REGION Network 14: Interface Signals 05 -Example: Model Flex-Pro-Line - IN/OUT- / Interface Signals 09
   // Aufruf des Schnittstellen Signal Bausteins Ba-Bereich 4 / Call the interface signals bool blocks of opmode 4
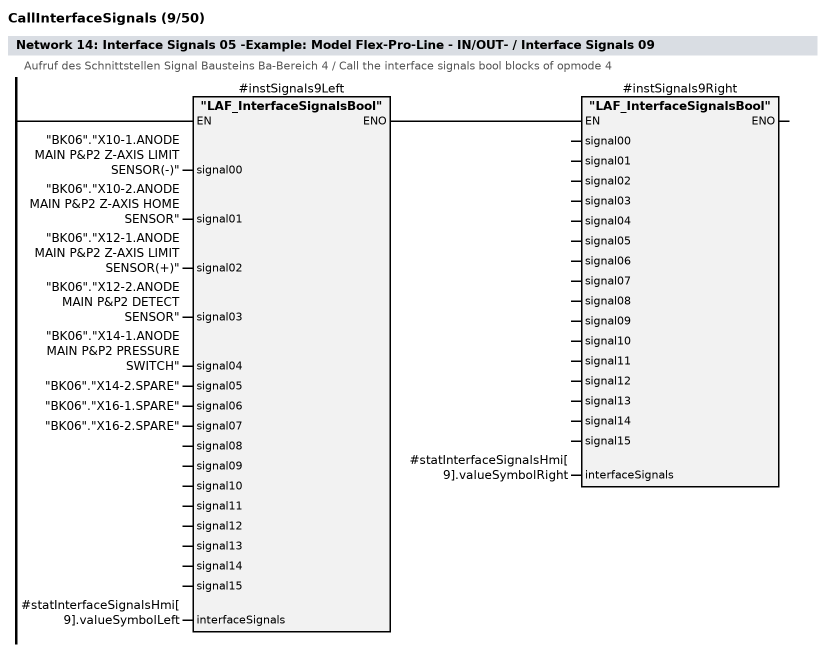
   RUNG wire#powerrail
      #instSignals9Left(signal00 := "BK06"."X10-1.ANODE MAIN P&P2 Z-AXIS LIMIT SENSOR(-)", signal01 := "BK06"."X10-2.ANODE MAIN P&P2 Z-AXIS HOME SENSOR", signal02 := "BK06"."X12-1.ANODE MAIN P&P2 Z-AXIS LIMIT SENSOR(+)", signal03 := "BK06"."X12-2.ANODE MAIN P&P2 DETECT SENSOR", signal04 := "BK06"."X14-1.ANODE MAIN P&P2 PRESSURE SWITCH", signal05 := "BK06"."X14-2.SPARE", signal06 := "BK06"."X16-1.SPARE", signal07 := "BK06"."X16-2.SPARE", signal08 :=, signal09 :=, signal10 :=, signal11 :=, signal12 :=, signal13 :=, signal14 :=, signal15 :=, interfaceSignals := #statInterfaceSignalsHmi[9].valueSymbolLeft)
      #instSignals9Right(signal00 :=, signal01 :=, signal02 :=, signal03 :=, signal04 :=, signal05 :=, signal06 :=, signal07 :=, signal08 :=, signal09 :=, signal10 :=, signal11 :=, signal12 :=, signal13 :=, signal14 :=, signal15 :=, interfaceSignals := #statInterfaceSignalsHmi[9].valueSymbolRight)
   END_RUNG
   // the same network as SCL:
   #instSignals9Left(signal00 := "BK06"."X10-1.ANODE MAIN P&P2 Z-AXIS LIMIT SENSOR(-)",   // "LAF_InterfaceSignalsBool"
                     signal01 := "BK06"."X10-2.ANODE MAIN P&P2 Z-AXIS HOME SENSOR",
                     signal02 := "BK06"."X12-1.ANODE MAIN P&P2 Z-AXIS LIMIT SENSOR(+)",
                     signal03 := "BK06"."X12-2.ANODE MAIN P&P2 DETECT SENSOR",
                     signal04 := "BK06"."X14-1.ANODE MAIN P&P2 PRESSURE SWITCH",
                     signal05 := "BK06"."X14-2.SPARE",
                     signal06 := "BK06"."X16-1.SPARE",
                     signal07 := "BK06"."X16-2.SPARE",
                     interfaceSignals := #statInterfaceSignalsHmi[9].valueSymbolLeft,
                     ENO => #_w1);
   IF #_w1 THEN
       #instSignals9Right(interfaceSignals := #statInterfaceSignalsHmi[9].valueSymbolRight);   // "LAF_InterfaceSignalsBool"
   END_IF;
END_REGION

REGION Network 15: Interface Signals 05 -Example: Model Flex-Pro-Line - IN/OUT- / Interface Signals 10
   // Aufruf des Schnittstellen Signal Bausteins Ba-Bereich 4 / Call the interface signals bool blocks of opmode 4
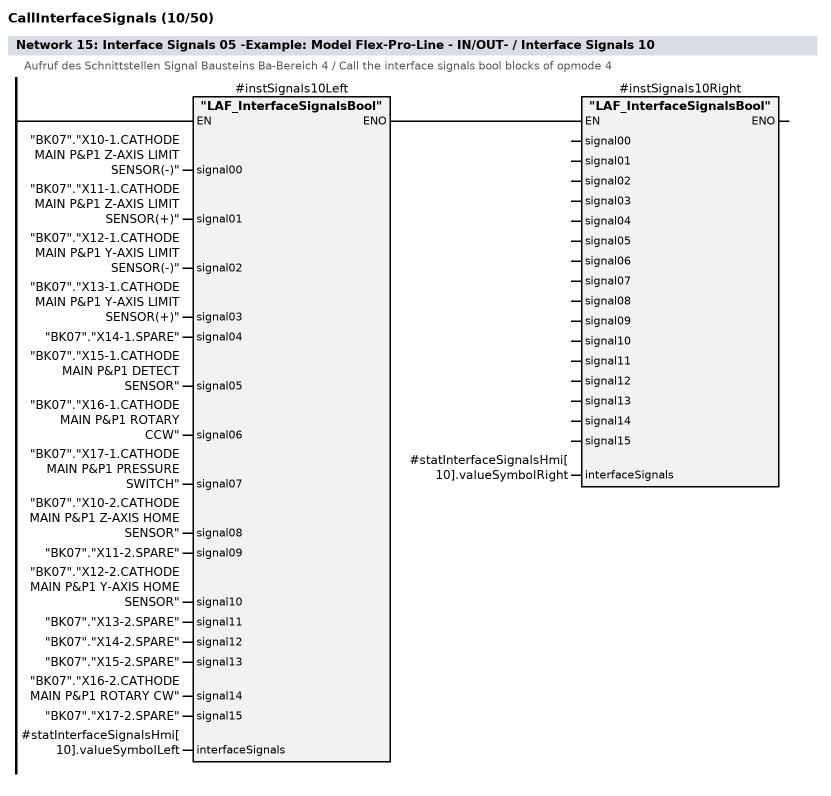
   RUNG wire#powerrail
      #instSignals10Left(signal00 := "BK07"."X10-1.CATHODE MAIN P&P1 Z-AXIS LIMIT SENSOR(-)", signal01 := "BK07"."X11-1.CATHODE MAIN P&P1 Z-AXIS LIMIT SENSOR(+)", signal02 := "BK07"."X12-1.CATHODE MAIN P&P1 Y-AXIS LIMIT SENSOR(-)", signal03 := "BK07"."X13-1.CATHODE MAIN P&P1 Y-AXIS LIMIT SENSOR(+)", signal04 := "BK07"."X14-1.SPARE", signal05 := "BK07"."X15-1.CATHODE MAIN P&P1 DETECT SENSOR", signal06 := "BK07"."X16-1.CATHODE MAIN P&P1 ROTARY CCW", signal07 := "BK07"."X17-1.CATHODE MAIN P&P1 PRESSURE SWITCH", signal08 := "BK07"."X10-2.CATHODE MAIN P&P1 Z-AXIS HOME SENSOR", signal09 := "BK07"."X11-2.SPARE", signal10 := "BK07"."X12-2.CATHODE MAIN P&P1 Y-AXIS HOME SENSOR", signal11 := "BK07"."X13-2.SPARE", signal12 := "BK07"."X14-2.SPARE", signal13 := "BK07"."X15-2.SPARE", signal14 := "BK07"."X16-2.CATHODE MAIN P&P1 ROTARY CW", signal15 := "BK07"."X17-2.SPARE", interfaceSignals := #statInterfaceSignalsHmi[10].valueSymbolLeft)
      #instSignals10Right(signal00 :=, signal01 :=, signal02 :=, signal03 :=, signal04 :=, signal05 :=, signal06 :=, signal07 :=, signal08 :=, signal09 :=, signal10 :=, signal11 :=, signal12 :=, signal13 :=, signal14 :=, signal15 :=, interfaceSignals := #statInterfaceSignalsHmi[10].valueSymbolRight)
   END_RUNG
   // the same network as SCL:
   #instSignals10Left(signal00 := "BK07"."X10-1.CATHODE MAIN P&P1 Z-AXIS LIMIT SENSOR(-)",   // "LAF_InterfaceSignalsBool"
                      signal01 := "BK07"."X11-1.CATHODE MAIN P&P1 Z-AXIS LIMIT SENSOR(+)",
                      signal02 := "BK07"."X12-1.CATHODE MAIN P&P1 Y-AXIS LIMIT SENSOR(-)",
                      signal03 := "BK07"."X13-1.CATHODE MAIN P&P1 Y-AXIS LIMIT SENSOR(+)",
                      signal04 := "BK07"."X14-1.SPARE",
                      signal05 := "BK07"."X15-1.CATHODE MAIN P&P1 DETECT SENSOR",
                      signal06 := "BK07"."X16-1.CATHODE MAIN P&P1 ROTARY CCW",
                      signal07 := "BK07"."X17-1.CATHODE MAIN P&P1 PRESSURE SWITCH",
                      signal08 := "BK07"."X10-2.CATHODE MAIN P&P1 Z-AXIS HOME SENSOR",
                      signal09 := "BK07"."X11-2.SPARE",
                      signal10 := "BK07"."X12-2.CATHODE MAIN P&P1 Y-AXIS HOME SENSOR",
                      signal11 := "BK07"."X13-2.SPARE",
                      signal12 := "BK07"."X14-2.SPARE",
                      signal13 := "BK07"."X15-2.SPARE",
                      signal14 := "BK07"."X16-2.CATHODE MAIN P&P1 ROTARY CW",
                      signal15 := "BK07"."X17-2.SPARE",
                      interfaceSignals := #statInterfaceSignalsHmi[10].valueSymbolLeft,
                      ENO => #_w1);
   IF #_w1 THEN
       #instSignals10Right(interfaceSignals := #statInterfaceSignalsHmi[10].valueSymbolRight);   // "LAF_InterfaceSignalsBool"
   END_IF;
END_REGION

REGION Network 16: Interface Signals 05 -Example: Model Flex-Pro-Line - IN/OUT- / Interface Signals 11
   // Aufruf des Schnittstellen Signal Bausteins Ba-Bereich 4 / Call the interface signals bool blocks of opmode 4
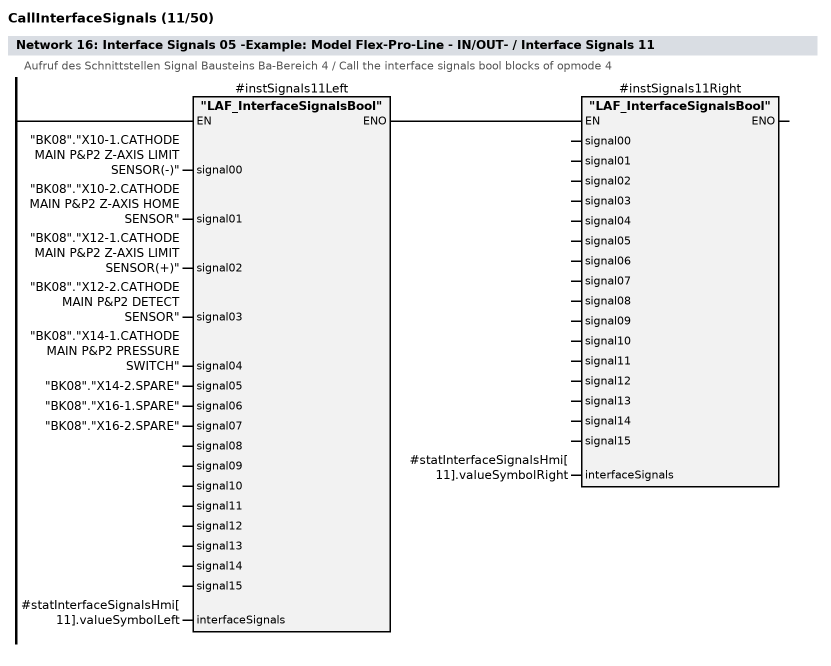
   RUNG wire#powerrail
      #instSignals11Left(signal00 := "BK08"."X10-1.CATHODE MAIN P&P2 Z-AXIS LIMIT SENSOR(-)", signal01 := "BK08"."X10-2.CATHODE MAIN P&P2 Z-AXIS HOME SENSOR", signal02 := "BK08"."X12-1.CATHODE MAIN P&P2 Z-AXIS LIMIT SENSOR(+)", signal03 := "BK08"."X12-2.CATHODE MAIN P&P2 DETECT SENSOR", signal04 := "BK08"."X14-1.CATHODE MAIN P&P2 PRESSURE SWITCH", signal05 := "BK08"."X14-2.SPARE", signal06 := "BK08"."X16-1.SPARE", signal07 := "BK08"."X16-2.SPARE", signal08 :=, signal09 :=, signal10 :=, signal11 :=, signal12 :=, signal13 :=, signal14 :=, signal15 :=, interfaceSignals := #statInterfaceSignalsHmi[11].valueSymbolLeft)
      #instSignals11Right(signal00 :=, signal01 :=, signal02 :=, signal03 :=, signal04 :=, signal05 :=, signal06 :=, signal07 :=, signal08 :=, signal09 :=, signal10 :=, signal11 :=, signal12 :=, signal13 :=, signal14 :=, signal15 :=, interfaceSignals := #statInterfaceSignalsHmi[11].valueSymbolRight)
   END_RUNG
   // the same network as SCL:
   #instSignals11Left(signal00 := "BK08"."X10-1.CATHODE MAIN P&P2 Z-AXIS LIMIT SENSOR(-)",   // "LAF_InterfaceSignalsBool"
                      signal01 := "BK08"."X10-2.CATHODE MAIN P&P2 Z-AXIS HOME SENSOR",
                      signal02 := "BK08"."X12-1.CATHODE MAIN P&P2 Z-AXIS LIMIT SENSOR(+)",
                      signal03 := "BK08"."X12-2.CATHODE MAIN P&P2 DETECT SENSOR",
                      signal04 := "BK08"."X14-1.CATHODE MAIN P&P2 PRESSURE SWITCH",
                      signal05 := "BK08"."X14-2.SPARE",
                      signal06 := "BK08"."X16-1.SPARE",
                      signal07 := "BK08"."X16-2.SPARE",
                      interfaceSignals := #statInterfaceSignalsHmi[11].valueSymbolLeft,
                      ENO => #_w1);
   IF #_w1 THEN
       #instSignals11Right(interfaceSignals := #statInterfaceSignalsHmi[11].valueSymbolRight);   // "LAF_InterfaceSignalsBool"
   END_IF;
END_REGION

REGION Network 17: Interface Signals 05 -Example: Model Flex-Pro-Line - IN/OUT- / Interface Signals 12
   // Aufruf des Schnittstellen Signal Bausteins Ba-Bereich 4 / Call the interface signals bool blocks of opmode 4
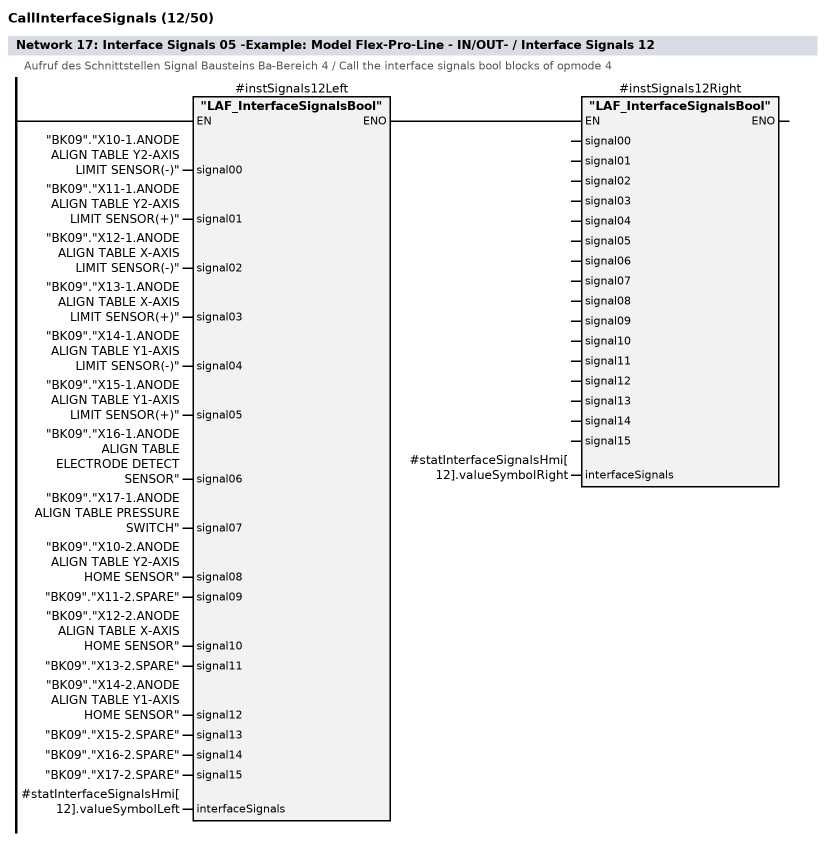
   RUNG wire#powerrail
      #instSignals12Left(signal00 := "BK09"."X10-1.ANODE ALIGN TABLE Y2-AXIS LIMIT SENSOR(-)", signal01 := "BK09"."X11-1.ANODE ALIGN TABLE Y2-AXIS LIMIT SENSOR(+)", signal02 := "BK09"."X12-1.ANODE ALIGN TABLE X-AXIS LIMIT SENSOR(-)", signal03 := "BK09"."X13-1.ANODE ALIGN TABLE X-AXIS LIMIT SENSOR(+)", signal04 := "BK09"."X14-1.ANODE ALIGN TABLE Y1-AXIS LIMIT SENSOR(-)", signal05 := "BK09"."X15-1.ANODE ALIGN TABLE Y1-AXIS LIMIT SENSOR(+)", signal06 := "BK09"."X16-1.ANODE ALIGN TABLE ELECTRODE DETECT SENSOR", signal07 := "BK09"."X17-1.ANODE ALIGN TABLE PRESSURE SWITCH", signal08 := "BK09"."X10-2.ANODE ALIGN TABLE Y2-AXIS HOME SENSOR", signal09 := "BK09"."X11-2.SPARE", signal10 := "BK09"."X12-2.ANODE ALIGN TABLE X-AXIS HOME SENSOR", signal11 := "BK09"."X13-2.SPARE", signal12 := "BK09"."X14-2.ANODE ALIGN TABLE Y1-AXIS HOME SENSOR", signal13 := "BK09"."X15-2.SPARE", signal14 := "BK09"."X16-2.SPARE", signal15 := "BK09"."X17-2.SPARE", interfaceSignals := #statInterfaceSignalsHmi[12].valueSymbolLeft)
      #instSignals12Right(signal00 :=, signal01 :=, signal02 :=, signal03 :=, signal04 :=, signal05 :=, signal06 :=, signal07 :=, signal08 :=, signal09 :=, signal10 :=, signal11 :=, signal12 :=, signal13 :=, signal14 :=, signal15 :=, interfaceSignals := #statInterfaceSignalsHmi[12].valueSymbolRight)
   END_RUNG
   // the same network as SCL:
   #instSignals12Left(signal00 := "BK09"."X10-1.ANODE ALIGN TABLE Y2-AXIS LIMIT SENSOR(-)",   // "LAF_InterfaceSignalsBool"
                      signal01 := "BK09"."X11-1.ANODE ALIGN TABLE Y2-AXIS LIMIT SENSOR(+)",
                      signal02 := "BK09"."X12-1.ANODE ALIGN TABLE X-AXIS LIMIT SENSOR(-)",
                      signal03 := "BK09"."X13-1.ANODE ALIGN TABLE X-AXIS LIMIT SENSOR(+)",
                      signal04 := "BK09"."X14-1.ANODE ALIGN TABLE Y1-AXIS LIMIT SENSOR(-)",
                      signal05 := "BK09"."X15-1.ANODE ALIGN TABLE Y1-AXIS LIMIT SENSOR(+)",
                      signal06 := "BK09"."X16-1.ANODE ALIGN TABLE ELECTRODE DETECT SENSOR",
                      signal07 := "BK09"."X17-1.ANODE ALIGN TABLE PRESSURE SWITCH",
                      signal08 := "BK09"."X10-2.ANODE ALIGN TABLE Y2-AXIS HOME SENSOR",
                      signal09 := "BK09"."X11-2.SPARE",
                      signal10 := "BK09"."X12-2.ANODE ALIGN TABLE X-AXIS HOME SENSOR",
                      signal11 := "BK09"."X13-2.SPARE",
                      signal12 := "BK09"."X14-2.ANODE ALIGN TABLE Y1-AXIS HOME SENSOR",
                      signal13 := "BK09"."X15-2.SPARE",
                      signal14 := "BK09"."X16-2.SPARE",
                      signal15 := "BK09"."X17-2.SPARE",
                      interfaceSignals := #statInterfaceSignalsHmi[12].valueSymbolLeft,
                      ENO => #_w1);
   IF #_w1 THEN
       #instSignals12Right(interfaceSignals := #statInterfaceSignalsHmi[12].valueSymbolRight);   // "LAF_InterfaceSignalsBool"
   END_IF;
END_REGION

REGION Network 18: Interface Signals 03 -Example: System flags & Clock flags- / Interface Signals13
   // Aufruf des Schnittstellen Signal Bausteins für die Systemvariablen / Call the interface signals bool blocks of system tags
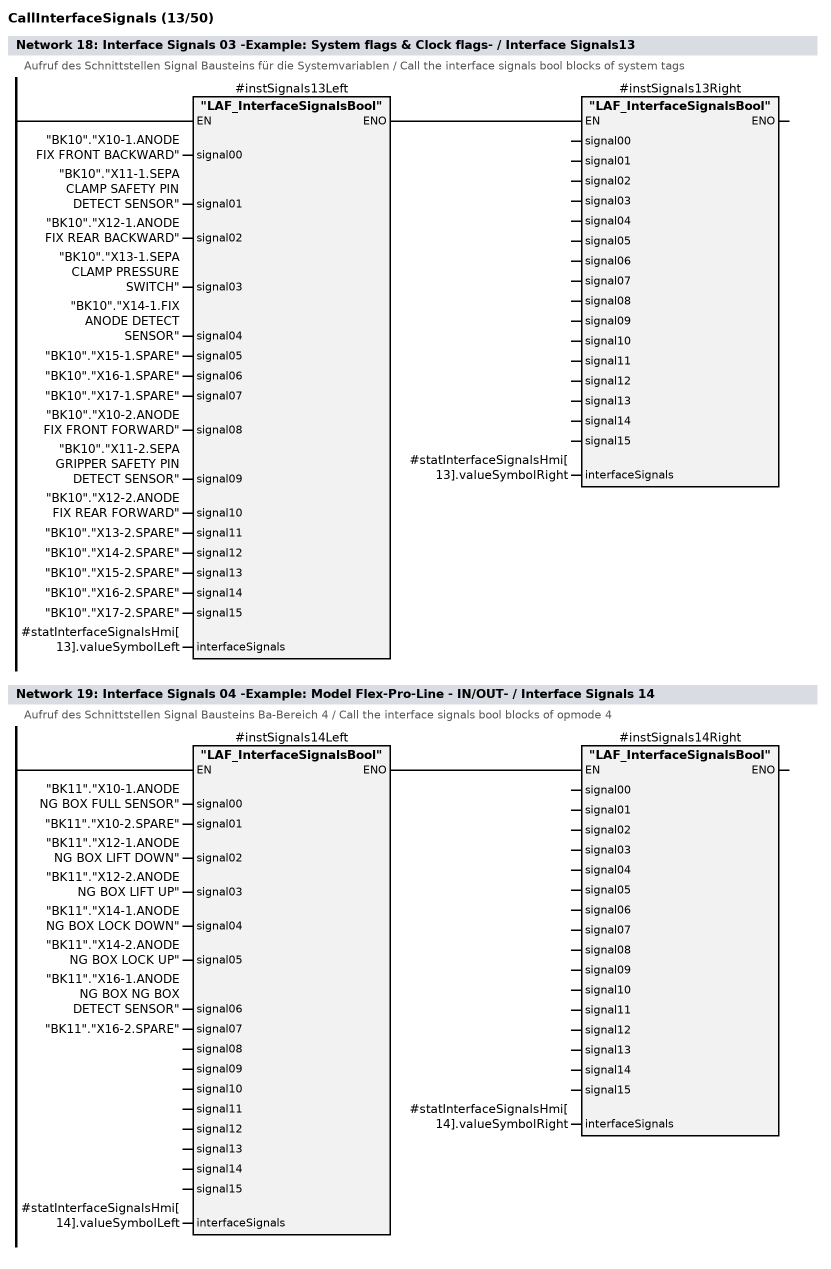
   RUNG wire#powerrail
      #instSignals13Left(signal00 := "BK10"."X10-1.ANODE FIX FRONT BACKWARD", signal01 := "BK10"."X11-1.SEPA CLAMP SAFETY PIN DETECT SENSOR", signal02 := "BK10"."X12-1.ANODE FIX REAR BACKWARD", signal03 := "BK10"."X13-1.SEPA CLAMP PRESSURE SWITCH", signal04 := "BK10"."X14-1.FIX ANODE DETECT SENSOR", signal05 := "BK10"."X15-1.SPARE", signal06 := "BK10"."X16-1.SPARE", signal07 := "BK10"."X17-1.SPARE", signal08 := "BK10"."X10-2.ANODE FIX FRONT FORWARD", signal09 := "BK10"."X11-2.SEPA GRIPPER SAFETY PIN DETECT SENSOR", signal10 := "BK10"."X12-2.ANODE FIX REAR FORWARD", signal11 := "BK10"."X13-2.SPARE", signal12 := "BK10"."X14-2.SPARE", signal13 := "BK10"."X15-2.SPARE", signal14 := "BK10"."X16-2.SPARE", signal15 := "BK10"."X17-2.SPARE", interfaceSignals := #statInterfaceSignalsHmi[13].valueSymbolLeft)
      #instSignals13Right(signal00 :=, signal01 :=, signal02 :=, signal03 :=, signal04 :=, signal05 :=, signal06 :=, signal07 :=, signal08 :=, signal09 :=, signal10 :=, signal11 :=, signal12 :=, signal13 :=, signal14 :=, signal15 :=, interfaceSignals := #statInterfaceSignalsHmi[13].valueSymbolRight)
   END_RUNG
   // the same network as SCL:
   #instSignals13Left(signal00 := "BK10"."X10-1.ANODE FIX FRONT BACKWARD",   // "LAF_InterfaceSignalsBool"
                      signal01 := "BK10"."X11-1.SEPA CLAMP SAFETY PIN DETECT SENSOR",
                      signal02 := "BK10"."X12-1.ANODE FIX REAR BACKWARD",
                      signal03 := "BK10"."X13-1.SEPA CLAMP PRESSURE SWITCH",
                      signal04 := "BK10"."X14-1.FIX ANODE DETECT SENSOR",
                      signal05 := "BK10"."X15-1.SPARE",
                      signal06 := "BK10"."X16-1.SPARE",
                      signal07 := "BK10"."X17-1.SPARE",
                      signal08 := "BK10"."X10-2.ANODE FIX FRONT FORWARD",
                      signal09 := "BK10"."X11-2.SEPA GRIPPER SAFETY PIN DETECT SENSOR",
                      signal10 := "BK10"."X12-2.ANODE FIX REAR FORWARD",
                      signal11 := "BK10"."X13-2.SPARE",
                      signal12 := "BK10"."X14-2.SPARE",
                      signal13 := "BK10"."X15-2.SPARE",
                      signal14 := "BK10"."X16-2.SPARE",
                      signal15 := "BK10"."X17-2.SPARE",
                      interfaceSignals := #statInterfaceSignalsHmi[13].valueSymbolLeft,
                      ENO => #_w1);
   IF #_w1 THEN
       #instSignals13Right(interfaceSignals := #statInterfaceSignalsHmi[13].valueSymbolRight);   // "LAF_InterfaceSignalsBool"
   END_IF;
END_REGION

REGION Network 19: Interface Signals 04 -Example: Model Flex-Pro-Line - IN/OUT- / Interface Signals 14
   // Aufruf des Schnittstellen Signal Bausteins Ba-Bereich 4 / Call the interface signals bool blocks of opmode 4
   RUNG wire#powerrail
      #instSignals14Left(signal00 := "BK11"."X10-1.ANODE NG BOX FULL SENSOR", signal01 := "BK11"."X10-2.SPARE", signal02 := "BK11"."X12-1.ANODE NG BOX LIFT DOWN", signal03 := "BK11"."X12-2.ANODE NG BOX LIFT UP", signal04 := "BK11"."X14-1.ANODE NG BOX LOCK DOWN", signal05 := "BK11"."X14-2.ANODE NG BOX LOCK UP", signal06 := "BK11"."X16-1.ANODE NG BOX NG BOX DETECT SENSOR", signal07 := "BK11"."X16-2.SPARE", signal08 :=, signal09 :=, signal10 :=, signal11 :=, signal12 :=, signal13 :=, signal14 :=, signal15 :=, interfaceSignals := #statInterfaceSignalsHmi[14].valueSymbolLeft)
      #instSignals14Right(signal00 :=, signal01 :=, signal02 :=, signal03 :=, signal04 :=, signal05 :=, signal06 :=, signal07 :=, signal08 :=, signal09 :=, signal10 :=, signal11 :=, signal12 :=, signal13 :=, signal14 :=, signal15 :=, interfaceSignals := #statInterfaceSignalsHmi[14].valueSymbolRight)
   END_RUNG
   // the same network as SCL:
   #instSignals14Left(signal00 := "BK11"."X10-1.ANODE NG BOX FULL SENSOR",   // "LAF_InterfaceSignalsBool"
                      signal01 := "BK11"."X10-2.SPARE",
                      signal02 := "BK11"."X12-1.ANODE NG BOX LIFT DOWN",
                      signal03 := "BK11"."X12-2.ANODE NG BOX LIFT UP",
                      signal04 := "BK11"."X14-1.ANODE NG BOX LOCK DOWN",
                      signal05 := "BK11"."X14-2.ANODE NG BOX LOCK UP",
                      signal06 := "BK11"."X16-1.ANODE NG BOX NG BOX DETECT SENSOR",
                      signal07 := "BK11"."X16-2.SPARE",
                      interfaceSignals := #statInterfaceSignalsHmi[14].valueSymbolLeft,
                      ENO => #_w1);
   IF #_w1 THEN
       #instSignals14Right(interfaceSignals := #statInterfaceSignalsHmi[14].valueSymbolRight);   // "LAF_InterfaceSignalsBool"
   END_IF;
END_REGION

REGION Network 20: Interface Signals 05 -Example: Model Flex-Pro-Line - IN/OUT- / Interface Signals 15
   // Aufruf des Schnittstellen Signal Bausteins Ba-Bereich 4 / Call the interface signals bool blocks of opmode 4
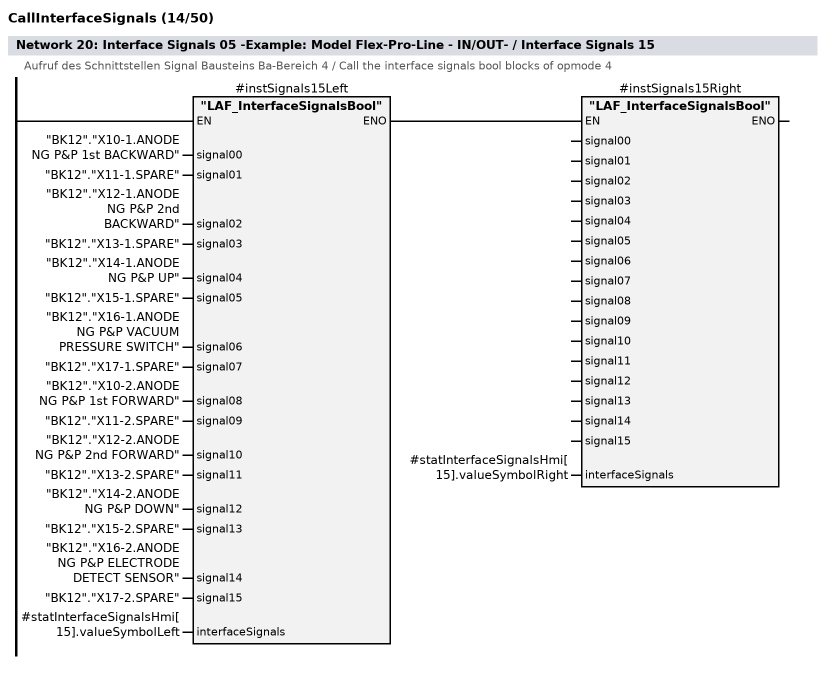
   RUNG wire#powerrail
      #instSignals15Left(signal00 := "BK12"."X10-1.ANODE NG P&P 1st BACKWARD", signal01 := "BK12"."X11-1.SPARE", signal02 := "BK12"."X12-1.ANODE NG P&P 2nd BACKWARD", signal03 := "BK12"."X13-1.SPARE", signal04 := "BK12"."X14-1.ANODE NG P&P UP", signal05 := "BK12"."X15-1.SPARE", signal06 := "BK12"."X16-1.ANODE NG P&P VACUUM PRESSURE SWITCH", signal07 := "BK12"."X17-1.SPARE", signal08 := "BK12"."X10-2.ANODE NG P&P 1st FORWARD", signal09 := "BK12"."X11-2.SPARE", signal10 := "BK12"."X12-2.ANODE NG P&P 2nd FORWARD", signal11 := "BK12"."X13-2.SPARE", signal12 := "BK12"."X14-2.ANODE NG P&P DOWN", signal13 := "BK12"."X15-2.SPARE", signal14 := "BK12"."X16-2.ANODE NG P&P ELECTRODE DETECT SENSOR", signal15 := "BK12"."X17-2.SPARE", interfaceSignals := #statInterfaceSignalsHmi[15].valueSymbolLeft)
      #instSignals15Right(signal00 :=, signal01 :=, signal02 :=, signal03 :=, signal04 :=, signal05 :=, signal06 :=, signal07 :=, signal08 :=, signal09 :=, signal10 :=, signal11 :=, signal12 :=, signal13 :=, signal14 :=, signal15 :=, interfaceSignals := #statInterfaceSignalsHmi[15].valueSymbolRight)
   END_RUNG
   // the same network as SCL:
   #instSignals15Left(signal00 := "BK12"."X10-1.ANODE NG P&P 1st BACKWARD",   // "LAF_InterfaceSignalsBool"
                      signal01 := "BK12"."X11-1.SPARE",
                      signal02 := "BK12"."X12-1.ANODE NG P&P 2nd BACKWARD",
                      signal03 := "BK12"."X13-1.SPARE",
                      signal04 := "BK12"."X14-1.ANODE NG P&P UP",
                      signal05 := "BK12"."X15-1.SPARE",
                      signal06 := "BK12"."X16-1.ANODE NG P&P VACUUM PRESSURE SWITCH",
                      signal07 := "BK12"."X17-1.SPARE",
                      signal08 := "BK12"."X10-2.ANODE NG P&P 1st FORWARD",
                      signal09 := "BK12"."X11-2.SPARE",
                      signal10 := "BK12"."X12-2.ANODE NG P&P 2nd FORWARD",
                      signal11 := "BK12"."X13-2.SPARE",
                      signal12 := "BK12"."X14-2.ANODE NG P&P DOWN",
                      signal13 := "BK12"."X15-2.SPARE",
                      signal14 := "BK12"."X16-2.ANODE NG P&P ELECTRODE DETECT SENSOR",
                      signal15 := "BK12"."X17-2.SPARE",
                      interfaceSignals := #statInterfaceSignalsHmi[15].valueSymbolLeft,
                      ENO => #_w1);
   IF #_w1 THEN
       #instSignals15Right(interfaceSignals := #statInterfaceSignalsHmi[15].valueSymbolRight);   // "LAF_InterfaceSignalsBool"
   END_IF;
END_REGION

REGION Network 21: Interface Signals 05 -Example: Model Flex-Pro-Line - IN/OUT- / Interface Signals 16
   // Aufruf des Schnittstellen Signal Bausteins Ba-Bereich 4 / Call the interface signals bool blocks of opmode 4
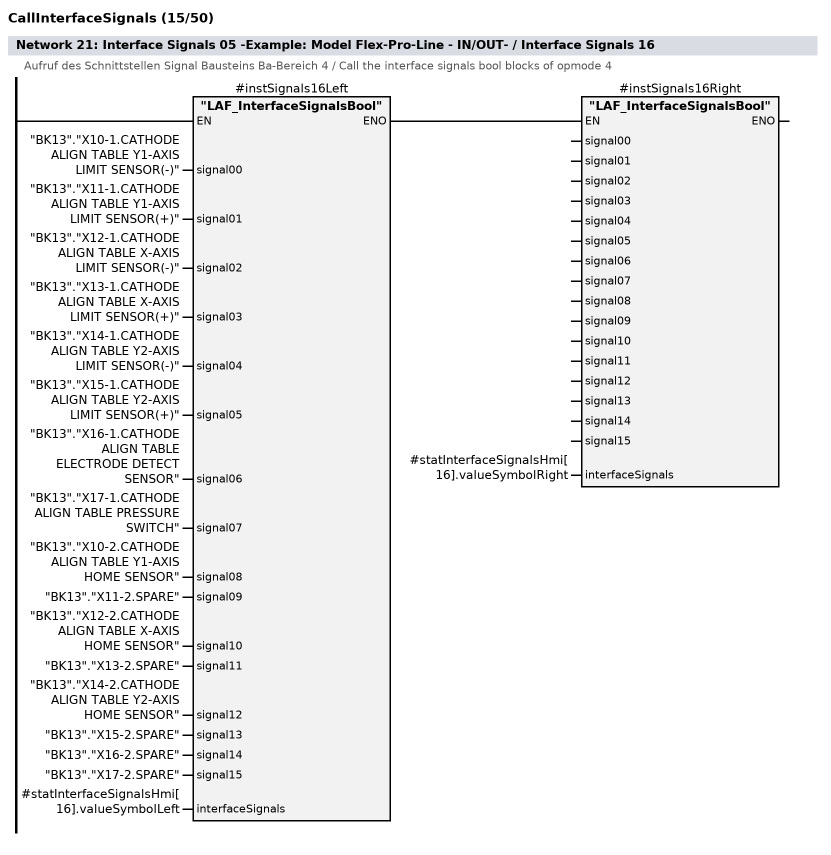
   RUNG wire#powerrail
      #instSignals16Left(signal00 := "BK13"."X10-1.CATHODE ALIGN TABLE Y1-AXIS LIMIT SENSOR(-)", signal01 := "BK13"."X11-1.CATHODE ALIGN TABLE Y1-AXIS LIMIT SENSOR(+)", signal02 := "BK13"."X12-1.CATHODE ALIGN TABLE X-AXIS LIMIT SENSOR(-)", signal03 := "BK13"."X13-1.CATHODE ALIGN TABLE X-AXIS LIMIT SENSOR(+)", signal04 := "BK13"."X14-1.CATHODE ALIGN TABLE Y2-AXIS LIMIT SENSOR(-)", signal05 := "BK13"."X15-1.CATHODE ALIGN TABLE Y2-AXIS LIMIT SENSOR(+)", signal06 := "BK13"."X16-1.CATHODE ALIGN TABLE ELECTRODE DETECT SENSOR", signal07 := "BK13"."X17-1.CATHODE ALIGN TABLE PRESSURE SWITCH", signal08 := "BK13"."X10-2.CATHODE ALIGN TABLE Y1-AXIS HOME SENSOR", signal09 := "BK13"."X11-2.SPARE", signal10 := "BK13"."X12-2.CATHODE ALIGN TABLE X-AXIS HOME SENSOR", signal11 := "BK13"."X13-2.SPARE", signal12 := "BK13"."X14-2.CATHODE ALIGN TABLE Y2-AXIS HOME SENSOR", signal13 := "BK13"."X15-2.SPARE", signal14 := "BK13"."X16-2.SPARE", signal15 := "BK13"."X17-2.SPARE", interfaceSignals := #statInterfaceSignalsHmi[16].valueSymbolLeft)
      #instSignals16Right(signal00 :=, signal01 :=, signal02 :=, signal03 :=, signal04 :=, signal05 :=, signal06 :=, signal07 :=, signal08 :=, signal09 :=, signal10 :=, signal11 :=, signal12 :=, signal13 :=, signal14 :=, signal15 :=, interfaceSignals := #statInterfaceSignalsHmi[16].valueSymbolRight)
   END_RUNG
   // the same network as SCL:
   #instSignals16Left(signal00 := "BK13"."X10-1.CATHODE ALIGN TABLE Y1-AXIS LIMIT SENSOR(-)",   // "LAF_InterfaceSignalsBool"
                      signal01 := "BK13"."X11-1.CATHODE ALIGN TABLE Y1-AXIS LIMIT SENSOR(+)",
                      signal02 := "BK13"."X12-1.CATHODE ALIGN TABLE X-AXIS LIMIT SENSOR(-)",
                      signal03 := "BK13"."X13-1.CATHODE ALIGN TABLE X-AXIS LIMIT SENSOR(+)",
                      signal04 := "BK13"."X14-1.CATHODE ALIGN TABLE Y2-AXIS LIMIT SENSOR(-)",
                      signal05 := "BK13"."X15-1.CATHODE ALIGN TABLE Y2-AXIS LIMIT SENSOR(+)",
                      signal06 := "BK13"."X16-1.CATHODE ALIGN TABLE ELECTRODE DETECT SENSOR",
                      signal07 := "BK13"."X17-1.CATHODE ALIGN TABLE PRESSURE SWITCH",
                      signal08 := "BK13"."X10-2.CATHODE ALIGN TABLE Y1-AXIS HOME SENSOR",
                      signal09 := "BK13"."X11-2.SPARE",
                      signal10 := "BK13"."X12-2.CATHODE ALIGN TABLE X-AXIS HOME SENSOR",
                      signal11 := "BK13"."X13-2.SPARE",
                      signal12 := "BK13"."X14-2.CATHODE ALIGN TABLE Y2-AXIS HOME SENSOR",
                      signal13 := "BK13"."X15-2.SPARE",
                      signal14 := "BK13"."X16-2.SPARE",
                      signal15 := "BK13"."X17-2.SPARE",
                      interfaceSignals := #statInterfaceSignalsHmi[16].valueSymbolLeft,
                      ENO => #_w1);
   IF #_w1 THEN
       #instSignals16Right(interfaceSignals := #statInterfaceSignalsHmi[16].valueSymbolRight);   // "LAF_InterfaceSignalsBool"
   END_IF;
END_REGION

REGION Network 22: Interface Signals 05 -Example: Model Flex-Pro-Line - IN/OUT- / Interface Signals 17
   // Aufruf des Schnittstellen Signal Bausteins Ba-Bereich 4 / Call the interface signals bool blocks of opmode 4
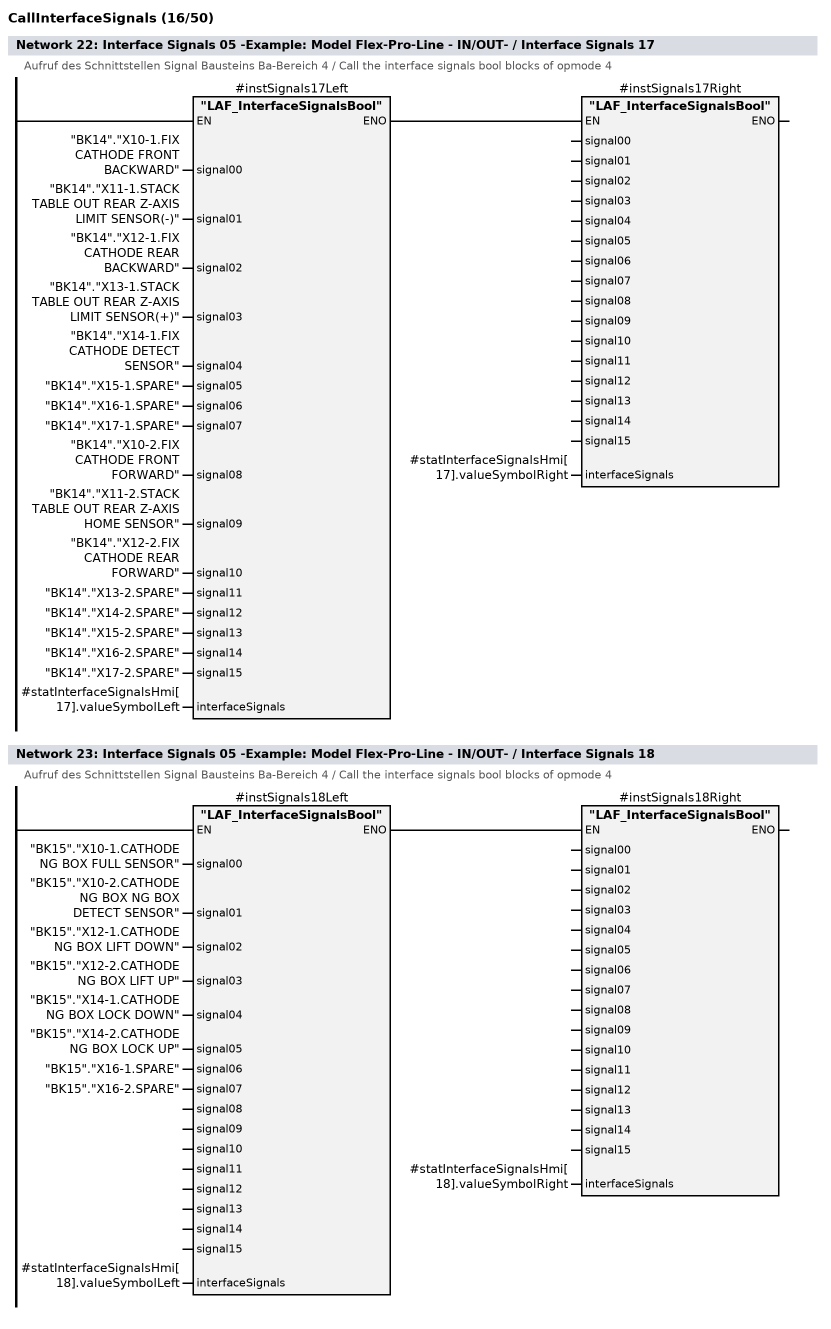
   RUNG wire#powerrail
      #instSignals17Left(signal00 := "BK14"."X10-1.FIX CATHODE FRONT BACKWARD", signal01 := "BK14"."X11-1.STACK TABLE OUT REAR Z-AXIS LIMIT SENSOR(-)", signal02 := "BK14"."X12-1.FIX CATHODE REAR BACKWARD", signal03 := "BK14"."X13-1.STACK TABLE OUT REAR Z-AXIS LIMIT SENSOR(+)", signal04 := "BK14"."X14-1.FIX CATHODE DETECT SENSOR", signal05 := "BK14"."X15-1.SPARE", signal06 := "BK14"."X16-1.SPARE", signal07 := "BK14"."X17-1.SPARE", signal08 := "BK14"."X10-2.FIX CATHODE FRONT FORWARD", signal09 := "BK14"."X11-2.STACK TABLE OUT REAR Z-AXIS HOME SENSOR", signal10 := "BK14"."X12-2.FIX CATHODE REAR FORWARD", signal11 := "BK14"."X13-2.SPARE", signal12 := "BK14"."X14-2.SPARE", signal13 := "BK14"."X15-2.SPARE", signal14 := "BK14"."X16-2.SPARE", signal15 := "BK14"."X17-2.SPARE", interfaceSignals := #statInterfaceSignalsHmi[17].valueSymbolLeft)
      #instSignals17Right(signal00 :=, signal01 :=, signal02 :=, signal03 :=, signal04 :=, signal05 :=, signal06 :=, signal07 :=, signal08 :=, signal09 :=, signal10 :=, signal11 :=, signal12 :=, signal13 :=, signal14 :=, signal15 :=, interfaceSignals := #statInterfaceSignalsHmi[17].valueSymbolRight)
   END_RUNG
   // the same network as SCL:
   #instSignals17Left(signal00 := "BK14"."X10-1.FIX CATHODE FRONT BACKWARD",   // "LAF_InterfaceSignalsBool"
                      signal01 := "BK14"."X11-1.STACK TABLE OUT REAR Z-AXIS LIMIT SENSOR(-)",
                      signal02 := "BK14"."X12-1.FIX CATHODE REAR BACKWARD",
                      signal03 := "BK14"."X13-1.STACK TABLE OUT REAR Z-AXIS LIMIT SENSOR(+)",
                      signal04 := "BK14"."X14-1.FIX CATHODE DETECT SENSOR",
                      signal05 := "BK14"."X15-1.SPARE",
                      signal06 := "BK14"."X16-1.SPARE",
                      signal07 := "BK14"."X17-1.SPARE",
                      signal08 := "BK14"."X10-2.FIX CATHODE FRONT FORWARD",
                      signal09 := "BK14"."X11-2.STACK TABLE OUT REAR Z-AXIS HOME SENSOR",
                      signal10 := "BK14"."X12-2.FIX CATHODE REAR FORWARD",
                      signal11 := "BK14"."X13-2.SPARE",
                      signal12 := "BK14"."X14-2.SPARE",
                      signal13 := "BK14"."X15-2.SPARE",
                      signal14 := "BK14"."X16-2.SPARE",
                      signal15 := "BK14"."X17-2.SPARE",
                      interfaceSignals := #statInterfaceSignalsHmi[17].valueSymbolLeft,
                      ENO => #_w1);
   IF #_w1 THEN
       #instSignals17Right(interfaceSignals := #statInterfaceSignalsHmi[17].valueSymbolRight);   // "LAF_InterfaceSignalsBool"
   END_IF;
END_REGION

REGION Network 23: Interface Signals 05 -Example: Model Flex-Pro-Line - IN/OUT- / Interface Signals 18
   // Aufruf des Schnittstellen Signal Bausteins Ba-Bereich 4 / Call the interface signals bool blocks of opmode 4
   RUNG wire#powerrail
      #instSignals18Left(signal00 := "BK15"."X10-1.CATHODE NG BOX FULL SENSOR", signal01 := "BK15"."X10-2.CATHODE NG BOX NG BOX DETECT SENSOR", signal02 := "BK15"."X12-1.CATHODE NG BOX LIFT DOWN", signal03 := "BK15"."X12-2.CATHODE NG BOX LIFT UP", signal04 := "BK15"."X14-1.CATHODE NG BOX LOCK DOWN", signal05 := "BK15"."X14-2.CATHODE NG BOX LOCK UP", signal06 := "BK15"."X16-1.SPARE", signal07 := "BK15"."X16-2.SPARE", signal08 :=, signal09 :=, signal10 :=, signal11 :=, signal12 :=, signal13 :=, signal14 :=, signal15 :=, interfaceSignals := #statInterfaceSignalsHmi[18].valueSymbolLeft)
      #instSignals18Right(signal00 :=, signal01 :=, signal02 :=, signal03 :=, signal04 :=, signal05 :=, signal06 :=, signal07 :=, signal08 :=, signal09 :=, signal10 :=, signal11 :=, signal12 :=, signal13 :=, signal14 :=, signal15 :=, interfaceSignals := #statInterfaceSignalsHmi[18].valueSymbolRight)
   END_RUNG
   // the same network as SCL:
   #instSignals18Left(signal00 := "BK15"."X10-1.CATHODE NG BOX FULL SENSOR",   // "LAF_InterfaceSignalsBool"
                      signal01 := "BK15"."X10-2.CATHODE NG BOX NG BOX DETECT SENSOR",
                      signal02 := "BK15"."X12-1.CATHODE NG BOX LIFT DOWN",
                      signal03 := "BK15"."X12-2.CATHODE NG BOX LIFT UP",
                      signal04 := "BK15"."X14-1.CATHODE NG BOX LOCK DOWN",
                      signal05 := "BK15"."X14-2.CATHODE NG BOX LOCK UP",
                      signal06 := "BK15"."X16-1.SPARE",
                      signal07 := "BK15"."X16-2.SPARE",
                      interfaceSignals := #statInterfaceSignalsHmi[18].valueSymbolLeft,
                      ENO => #_w1);
   IF #_w1 THEN
       #instSignals18Right(interfaceSignals := #statInterfaceSignalsHmi[18].valueSymbolRight);   // "LAF_InterfaceSignalsBool"
   END_IF;
END_REGION

REGION Network 24: Interface Signals 05 -Example: Model Flex-Pro-Line - IN/OUT- / Interface Signals 19
   // Aufruf des Schnittstellen Signal Bausteins Ba-Bereich 4 / Call the interface signals bool blocks of opmode 4
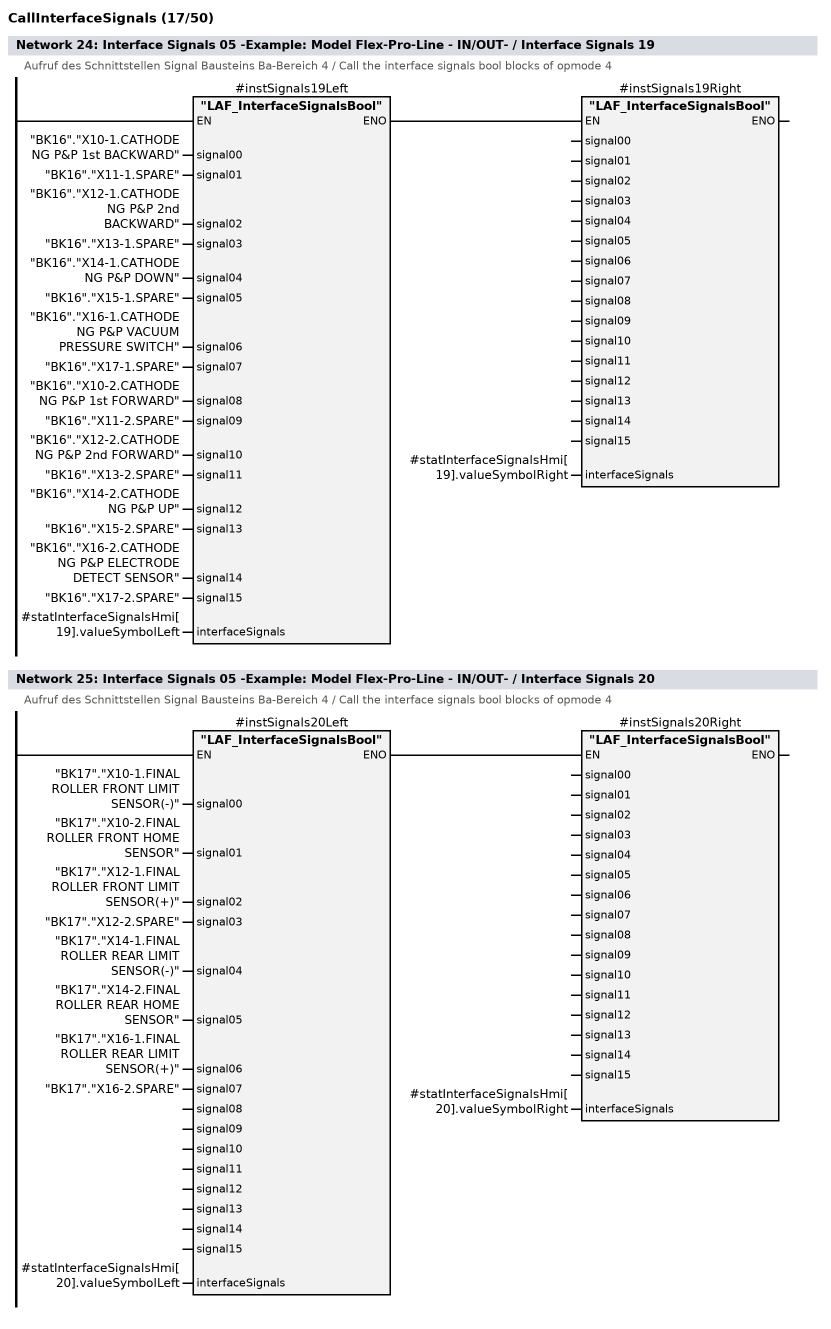
   RUNG wire#powerrail
      #instSignals19Left(signal00 := "BK16"."X10-1.CATHODE NG P&P 1st BACKWARD", signal01 := "BK16"."X11-1.SPARE", signal02 := "BK16"."X12-1.CATHODE NG P&P 2nd BACKWARD", signal03 := "BK16"."X13-1.SPARE", signal04 := "BK16"."X14-1.CATHODE NG P&P DOWN", signal05 := "BK16"."X15-1.SPARE", signal06 := "BK16"."X16-1.CATHODE NG P&P VACUUM PRESSURE SWITCH", signal07 := "BK16"."X17-1.SPARE", signal08 := "BK16"."X10-2.CATHODE NG P&P 1st FORWARD", signal09 := "BK16"."X11-2.SPARE", signal10 := "BK16"."X12-2.CATHODE NG P&P 2nd FORWARD", signal11 := "BK16"."X13-2.SPARE", signal12 := "BK16"."X14-2.CATHODE NG P&P UP", signal13 := "BK16"."X15-2.SPARE", signal14 := "BK16"."X16-2.CATHODE NG P&P ELECTRODE DETECT SENSOR", signal15 := "BK16"."X17-2.SPARE", interfaceSignals := #statInterfaceSignalsHmi[19].valueSymbolLeft)
      #instSignals19Right(signal00 :=, signal01 :=, signal02 :=, signal03 :=, signal04 :=, signal05 :=, signal06 :=, signal07 :=, signal08 :=, signal09 :=, signal10 :=, signal11 :=, signal12 :=, signal13 :=, signal14 :=, signal15 :=, interfaceSignals := #statInterfaceSignalsHmi[19].valueSymbolRight)
   END_RUNG
   // the same network as SCL:
   #instSignals19Left(signal00 := "BK16"."X10-1.CATHODE NG P&P 1st BACKWARD",   // "LAF_InterfaceSignalsBool"
                      signal01 := "BK16"."X11-1.SPARE",
                      signal02 := "BK16"."X12-1.CATHODE NG P&P 2nd BACKWARD",
                      signal03 := "BK16"."X13-1.SPARE",
                      signal04 := "BK16"."X14-1.CATHODE NG P&P DOWN",
                      signal05 := "BK16"."X15-1.SPARE",
                      signal06 := "BK16"."X16-1.CATHODE NG P&P VACUUM PRESSURE SWITCH",
                      signal07 := "BK16"."X17-1.SPARE",
                      signal08 := "BK16"."X10-2.CATHODE NG P&P 1st FORWARD",
                      signal09 := "BK16"."X11-2.SPARE",
                      signal10 := "BK16"."X12-2.CATHODE NG P&P 2nd FORWARD",
                      signal11 := "BK16"."X13-2.SPARE",
                      signal12 := "BK16"."X14-2.CATHODE NG P&P UP",
                      signal13 := "BK16"."X15-2.SPARE",
                      signal14 := "BK16"."X16-2.CATHODE NG P&P ELECTRODE DETECT SENSOR",
                      signal15 := "BK16"."X17-2.SPARE",
                      interfaceSignals := #statInterfaceSignalsHmi[19].valueSymbolLeft,
                      ENO => #_w1);
   IF #_w1 THEN
       #instSignals19Right(interfaceSignals := #statInterfaceSignalsHmi[19].valueSymbolRight);   // "LAF_InterfaceSignalsBool"
   END_IF;
END_REGION

REGION Network 25: Interface Signals 05 -Example: Model Flex-Pro-Line - IN/OUT- / Interface Signals 20
   // Aufruf des Schnittstellen Signal Bausteins Ba-Bereich 4 / Call the interface signals bool blocks of opmode 4
   RUNG wire#powerrail
      #instSignals20Left(signal00 := "BK17"."X10-1.FINAL ROLLER FRONT LIMIT SENSOR(-)", signal01 := "BK17"."X10-2.FINAL ROLLER FRONT HOME SENSOR", signal02 := "BK17"."X12-1.FINAL ROLLER FRONT LIMIT SENSOR(+)", signal03 := "BK17"."X12-2.SPARE", signal04 := "BK17"."X14-1.FINAL ROLLER REAR LIMIT SENSOR(-)", signal05 := "BK17"."X14-2.FINAL ROLLER REAR HOME SENSOR", signal06 := "BK17"."X16-1.FINAL ROLLER REAR LIMIT SENSOR(+)", signal07 := "BK17"."X16-2.SPARE", signal08 :=, signal09 :=, signal10 :=, signal11 :=, signal12 :=, signal13 :=, signal14 :=, signal15 :=, interfaceSignals := #statInterfaceSignalsHmi[20].valueSymbolLeft)
      #instSignals20Right(signal00 :=, signal01 :=, signal02 :=, signal03 :=, signal04 :=, signal05 :=, signal06 :=, signal07 :=, signal08 :=, signal09 :=, signal10 :=, signal11 :=, signal12 :=, signal13 :=, signal14 :=, signal15 :=, interfaceSignals := #statInterfaceSignalsHmi[20].valueSymbolRight)
   END_RUNG
   // the same network as SCL:
   #instSignals20Left(signal00 := "BK17"."X10-1.FINAL ROLLER FRONT LIMIT SENSOR(-)",   // "LAF_InterfaceSignalsBool"
                      signal01 := "BK17"."X10-2.FINAL ROLLER FRONT HOME SENSOR",
                      signal02 := "BK17"."X12-1.FINAL ROLLER FRONT LIMIT SENSOR(+)",
                      signal03 := "BK17"."X12-2.SPARE",
                      signal04 := "BK17"."X14-1.FINAL ROLLER REAR LIMIT SENSOR(-)",
                      signal05 := "BK17"."X14-2.FINAL ROLLER REAR HOME SENSOR",
                      signal06 := "BK17"."X16-1.FINAL ROLLER REAR LIMIT SENSOR(+)",
                      signal07 := "BK17"."X16-2.SPARE",
                      interfaceSignals := #statInterfaceSignalsHmi[20].valueSymbolLeft,
                      ENO => #_w1);
   IF #_w1 THEN
       #instSignals20Right(interfaceSignals := #statInterfaceSignalsHmi[20].valueSymbolRight);   // "LAF_InterfaceSignalsBool"
   END_IF;
END_REGION

REGION Network 26: Interface Signals 05 -Example: Model Flex-Pro-Line - IN/OUT- / Interface Signals 21
   // Aufruf des Schnittstellen Signal Bausteins Ba-Bereich 4 / Call the interface signals bool blocks of opmode 4
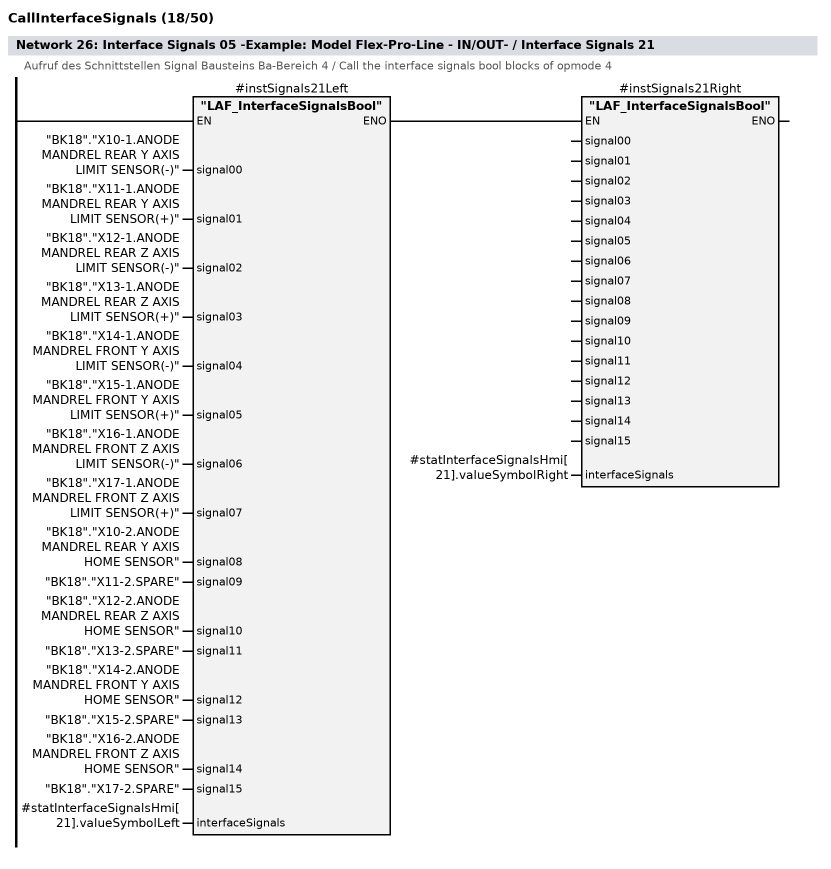
   RUNG wire#powerrail
      #instSignals21Left(signal00 := "BK18"."X10-1.ANODE MANDREL REAR Y AXIS LIMIT SENSOR(-)", signal01 := "BK18"."X11-1.ANODE MANDREL REAR Y AXIS LIMIT SENSOR(+)", signal02 := "BK18"."X12-1.ANODE MANDREL REAR Z AXIS LIMIT SENSOR(-)", signal03 := "BK18"."X13-1.ANODE MANDREL REAR Z AXIS LIMIT SENSOR(+)", signal04 := "BK18"."X14-1.ANODE MANDREL FRONT Y AXIS LIMIT SENSOR(-)", signal05 := "BK18"."X15-1.ANODE MANDREL FRONT Y AXIS LIMIT SENSOR(+)", signal06 := "BK18"."X16-1.ANODE MANDREL FRONT Z AXIS LIMIT SENSOR(-)", signal07 := "BK18"."X17-1.ANODE MANDREL FRONT Z AXIS LIMIT SENSOR(+)", signal08 := "BK18"."X10-2.ANODE MANDREL REAR Y AXIS HOME SENSOR", signal09 := "BK18"."X11-2.SPARE", signal10 := "BK18"."X12-2.ANODE MANDREL REAR Z AXIS HOME SENSOR", signal11 := "BK18"."X13-2.SPARE", signal12 := "BK18"."X14-2.ANODE MANDREL FRONT Y AXIS HOME SENSOR", signal13 := "BK18"."X15-2.SPARE", signal14 := "BK18"."X16-2.ANODE MANDREL FRONT Z AXIS HOME SENSOR", signal15 := "BK18"."X17-2.SPARE", interfaceSignals := #statInterfaceSignalsHmi[21].valueSymbolLeft)
      #instSignals21Right(signal00 :=, signal01 :=, signal02 :=, signal03 :=, signal04 :=, signal05 :=, signal06 :=, signal07 :=, signal08 :=, signal09 :=, signal10 :=, signal11 :=, signal12 :=, signal13 :=, signal14 :=, signal15 :=, interfaceSignals := #statInterfaceSignalsHmi[21].valueSymbolRight)
   END_RUNG
   // the same network as SCL:
   #instSignals21Left(signal00 := "BK18"."X10-1.ANODE MANDREL REAR Y AXIS LIMIT SENSOR(-)",   // "LAF_InterfaceSignalsBool"
                      signal01 := "BK18"."X11-1.ANODE MANDREL REAR Y AXIS LIMIT SENSOR(+)",
                      signal02 := "BK18"."X12-1.ANODE MANDREL REAR Z AXIS LIMIT SENSOR(-)",
                      signal03 := "BK18"."X13-1.ANODE MANDREL REAR Z AXIS LIMIT SENSOR(+)",
                      signal04 := "BK18"."X14-1.ANODE MANDREL FRONT Y AXIS LIMIT SENSOR(-)",
                      signal05 := "BK18"."X15-1.ANODE MANDREL FRONT Y AXIS LIMIT SENSOR(+)",
                      signal06 := "BK18"."X16-1.ANODE MANDREL FRONT Z AXIS LIMIT SENSOR(-)",
                      signal07 := "BK18"."X17-1.ANODE MANDREL FRONT Z AXIS LIMIT SENSOR(+)",
                      signal08 := "BK18"."X10-2.ANODE MANDREL REAR Y AXIS HOME SENSOR",
                      signal09 := "BK18"."X11-2.SPARE",
                      signal10 := "BK18"."X12-2.ANODE MANDREL REAR Z AXIS HOME SENSOR",
                      signal11 := "BK18"."X13-2.SPARE",
                      signal12 := "BK18"."X14-2.ANODE MANDREL FRONT Y AXIS HOME SENSOR",
                      signal13 := "BK18"."X15-2.SPARE",
                      signal14 := "BK18"."X16-2.ANODE MANDREL FRONT Z AXIS HOME SENSOR",
                      signal15 := "BK18"."X17-2.SPARE",
                      interfaceSignals := #statInterfaceSignalsHmi[21].valueSymbolLeft,
                      ENO => #_w1);
   IF #_w1 THEN
       #instSignals21Right(interfaceSignals := #statInterfaceSignalsHmi[21].valueSymbolRight);   // "LAF_InterfaceSignalsBool"
   END_IF;
END_REGION

REGION Network 27: Interface Signals 05 -Example: Model Flex-Pro-Line - IN/OUT- / Interface Signals 22
   // Aufruf des Schnittstellen Signal Bausteins Ba-Bereich 4 / Call the interface signals bool blocks of opmode 4
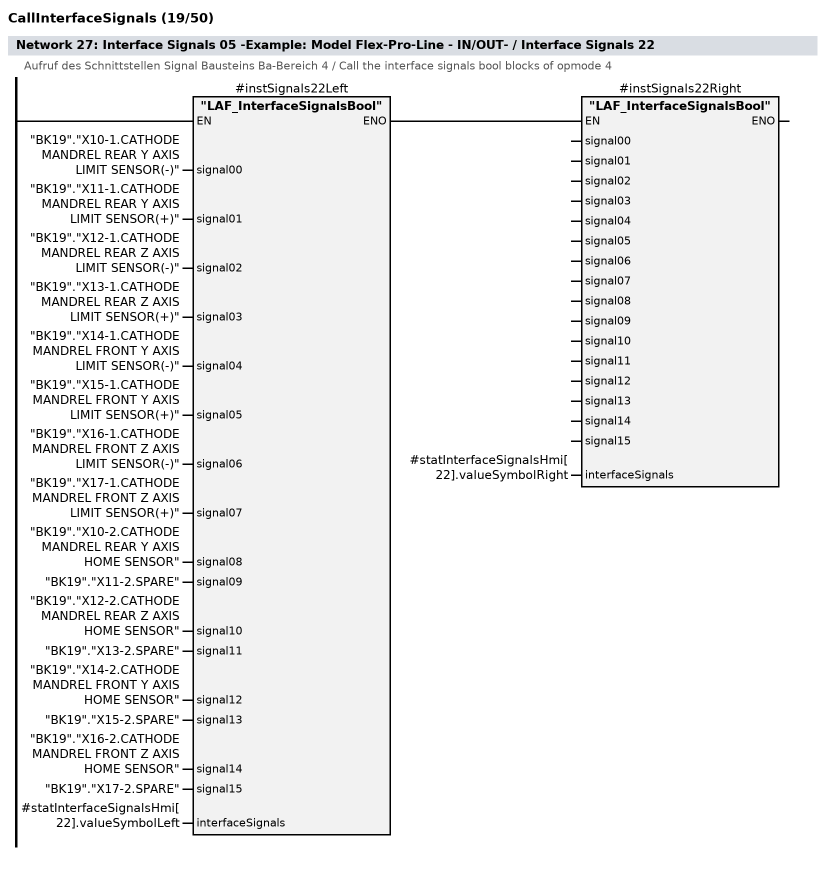
   RUNG wire#powerrail
      #instSignals22Left(signal00 := "BK19"."X10-1.CATHODE MANDREL REAR Y AXIS LIMIT SENSOR(-)", signal01 := "BK19"."X11-1.CATHODE MANDREL REAR Y AXIS LIMIT SENSOR(+)", signal02 := "BK19"."X12-1.CATHODE MANDREL REAR Z AXIS LIMIT SENSOR(-)", signal03 := "BK19"."X13-1.CATHODE MANDREL REAR Z AXIS LIMIT SENSOR(+)", signal04 := "BK19"."X14-1.CATHODE MANDREL FRONT Y AXIS LIMIT SENSOR(-)", signal05 := "BK19"."X15-1.CATHODE MANDREL FRONT Y AXIS LIMIT SENSOR(+)", signal06 := "BK19"."X16-1.CATHODE MANDREL FRONT Z AXIS LIMIT SENSOR(-)", signal07 := "BK19"."X17-1.CATHODE MANDREL FRONT Z AXIS LIMIT SENSOR(+)", signal08 := "BK19"."X10-2.CATHODE MANDREL REAR Y AXIS HOME SENSOR", signal09 := "BK19"."X11-2.SPARE", signal10 := "BK19"."X12-2.CATHODE MANDREL REAR Z AXIS HOME SENSOR", signal11 := "BK19"."X13-2.SPARE", signal12 := "BK19"."X14-2.CATHODE MANDREL FRONT Y AXIS HOME SENSOR", signal13 := "BK19"."X15-2.SPARE", signal14 := "BK19"."X16-2.CATHODE MANDREL FRONT Z AXIS HOME SENSOR", signal15 := "BK19"."X17-2.SPARE", interfaceSignals := #statInterfaceSignalsHmi[22].valueSymbolLeft)
      #instSignals22Right(signal00 :=, signal01 :=, signal02 :=, signal03 :=, signal04 :=, signal05 :=, signal06 :=, signal07 :=, signal08 :=, signal09 :=, signal10 :=, signal11 :=, signal12 :=, signal13 :=, signal14 :=, signal15 :=, interfaceSignals := #statInterfaceSignalsHmi[22].valueSymbolRight)
   END_RUNG
   // the same network as SCL:
   #instSignals22Left(signal00 := "BK19"."X10-1.CATHODE MANDREL REAR Y AXIS LIMIT SENSOR(-)",   // "LAF_InterfaceSignalsBool"
                      signal01 := "BK19"."X11-1.CATHODE MANDREL REAR Y AXIS LIMIT SENSOR(+)",
                      signal02 := "BK19"."X12-1.CATHODE MANDREL REAR Z AXIS LIMIT SENSOR(-)",
                      signal03 := "BK19"."X13-1.CATHODE MANDREL REAR Z AXIS LIMIT SENSOR(+)",
                      signal04 := "BK19"."X14-1.CATHODE MANDREL FRONT Y AXIS LIMIT SENSOR(-)",
                      signal05 := "BK19"."X15-1.CATHODE MANDREL FRONT Y AXIS LIMIT SENSOR(+)",
                      signal06 := "BK19"."X16-1.CATHODE MANDREL FRONT Z AXIS LIMIT SENSOR(-)",
                      signal07 := "BK19"."X17-1.CATHODE MANDREL FRONT Z AXIS LIMIT SENSOR(+)",
                      signal08 := "BK19"."X10-2.CATHODE MANDREL REAR Y AXIS HOME SENSOR",
                      signal09 := "BK19"."X11-2.SPARE",
                      signal10 := "BK19"."X12-2.CATHODE MANDREL REAR Z AXIS HOME SENSOR",
                      signal11 := "BK19"."X13-2.SPARE",
                      signal12 := "BK19"."X14-2.CATHODE MANDREL FRONT Y AXIS HOME SENSOR",
                      signal13 := "BK19"."X15-2.SPARE",
                      signal14 := "BK19"."X16-2.CATHODE MANDREL FRONT Z AXIS HOME SENSOR",
                      signal15 := "BK19"."X17-2.SPARE",
                      interfaceSignals := #statInterfaceSignalsHmi[22].valueSymbolLeft,
                      ENO => #_w1);
   IF #_w1 THEN
       #instSignals22Right(interfaceSignals := #statInterfaceSignalsHmi[22].valueSymbolRight);   // "LAF_InterfaceSignalsBool"
   END_IF;
END_REGION

REGION Network 28: Interface Signals 03 -Example: System flags & Clock flags- / Interface Signals23
   // Aufruf des Schnittstellen Signal Bausteins für die Systemvariablen / Call the interface signals bool blocks of system tags
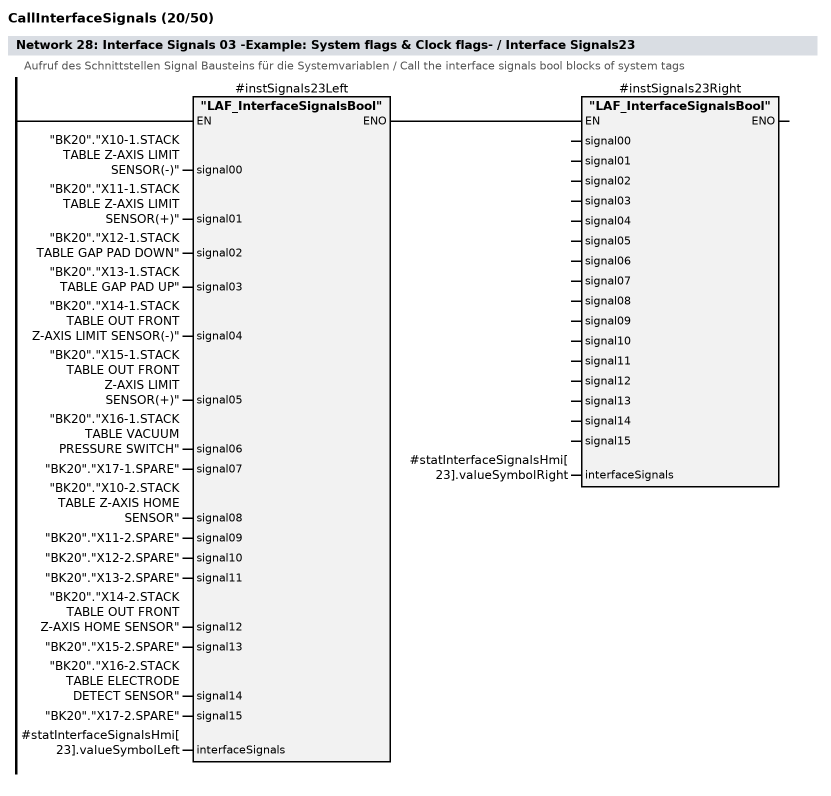
   RUNG wire#powerrail
      #instSignals23Left(signal00 := "BK20"."X10-1.STACK TABLE Z-AXIS LIMIT SENSOR(-)", signal01 := "BK20"."X11-1.STACK TABLE Z-AXIS LIMIT SENSOR(+)", signal02 := "BK20"."X12-1.STACK TABLE GAP PAD DOWN", signal03 := "BK20"."X13-1.STACK TABLE GAP PAD UP", signal04 := "BK20"."X14-1.STACK TABLE OUT FRONT Z-AXIS LIMIT SENSOR(-)", signal05 := "BK20"."X15-1.STACK TABLE OUT FRONT Z-AXIS LIMIT SENSOR(+)", signal06 := "BK20"."X16-1.STACK TABLE VACUUM PRESSURE SWITCH", signal07 := "BK20"."X17-1.SPARE", signal08 := "BK20"."X10-2.STACK TABLE Z-AXIS HOME SENSOR", signal09 := "BK20"."X11-2.SPARE", signal10 := "BK20"."X12-2.SPARE", signal11 := "BK20"."X13-2.SPARE", signal12 := "BK20"."X14-2.STACK TABLE OUT FRONT Z-AXIS HOME SENSOR", signal13 := "BK20"."X15-2.SPARE", signal14 := "BK20"."X16-2.STACK TABLE ELECTRODE DETECT SENSOR", signal15 := "BK20"."X17-2.SPARE", interfaceSignals := #statInterfaceSignalsHmi[23].valueSymbolLeft)
      #instSignals23Right(signal00 :=, signal01 :=, signal02 :=, signal03 :=, signal04 :=, signal05 :=, signal06 :=, signal07 :=, signal08 :=, signal09 :=, signal10 :=, signal11 :=, signal12 :=, signal13 :=, signal14 :=, signal15 :=, interfaceSignals := #statInterfaceSignalsHmi[23].valueSymbolRight)
   END_RUNG
   // the same network as SCL:
   #instSignals23Left(signal00 := "BK20"."X10-1.STACK TABLE Z-AXIS LIMIT SENSOR(-)",   // "LAF_InterfaceSignalsBool"
                      signal01 := "BK20"."X11-1.STACK TABLE Z-AXIS LIMIT SENSOR(+)",
                      signal02 := "BK20"."X12-1.STACK TABLE GAP PAD DOWN",
                      signal03 := "BK20"."X13-1.STACK TABLE GAP PAD UP",
                      signal04 := "BK20"."X14-1.STACK TABLE OUT FRONT Z-AXIS LIMIT SENSOR(-)",
                      signal05 := "BK20"."X15-1.STACK TABLE OUT FRONT Z-AXIS LIMIT SENSOR(+)",
                      signal06 := "BK20"."X16-1.STACK TABLE VACUUM PRESSURE SWITCH",
                      signal07 := "BK20"."X17-1.SPARE",
                      signal08 := "BK20"."X10-2.STACK TABLE Z-AXIS HOME SENSOR",
                      signal09 := "BK20"."X11-2.SPARE",
                      signal10 := "BK20"."X12-2.SPARE",
                      signal11 := "BK20"."X13-2.SPARE",
                      signal12 := "BK20"."X14-2.STACK TABLE OUT FRONT Z-AXIS HOME SENSOR",
                      signal13 := "BK20"."X15-2.SPARE",
                      signal14 := "BK20"."X16-2.STACK TABLE ELECTRODE DETECT SENSOR",
                      signal15 := "BK20"."X17-2.SPARE",
                      interfaceSignals := #statInterfaceSignalsHmi[23].valueSymbolLeft,
                      ENO => #_w1);
   IF #_w1 THEN
       #instSignals23Right(interfaceSignals := #statInterfaceSignalsHmi[23].valueSymbolRight);   // "LAF_InterfaceSignalsBool"
   END_IF;
END_REGION

REGION Network 29: Interface Signals 04 -Example: Model Flex-Pro-Line - IN/OUT- / Interface Signals 24
   // Aufruf des Schnittstellen Signal Bausteins Ba-Bereich 4 / Call the interface signals bool blocks of opmode 4
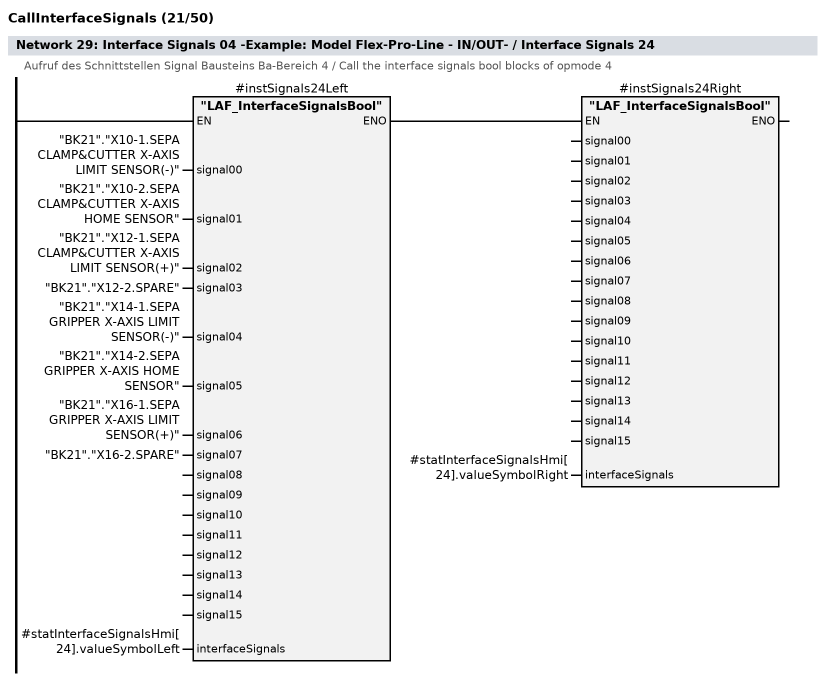
   RUNG wire#powerrail
      #instSignals24Left(signal00 := "BK21"."X10-1.SEPA CLAMP&CUTTER X-AXIS LIMIT SENSOR(-)", signal01 := "BK21"."X10-2.SEPA CLAMP&CUTTER X-AXIS HOME SENSOR", signal02 := "BK21"."X12-1.SEPA CLAMP&CUTTER X-AXIS LIMIT SENSOR(+)", signal03 := "BK21"."X12-2.SPARE", signal04 := "BK21"."X14-1.SEPA GRIPPER X-AXIS LIMIT SENSOR(-)", signal05 := "BK21"."X14-2.SEPA GRIPPER X-AXIS HOME SENSOR", signal06 := "BK21"."X16-1.SEPA GRIPPER X-AXIS LIMIT SENSOR(+)", signal07 := "BK21"."X16-2.SPARE", signal08 :=, signal09 :=, signal10 :=, signal11 :=, signal12 :=, signal13 :=, signal14 :=, signal15 :=, interfaceSignals := #statInterfaceSignalsHmi[24].valueSymbolLeft)
      #instSignals24Right(signal00 :=, signal01 :=, signal02 :=, signal03 :=, signal04 :=, signal05 :=, signal06 :=, signal07 :=, signal08 :=, signal09 :=, signal10 :=, signal11 :=, signal12 :=, signal13 :=, signal14 :=, signal15 :=, interfaceSignals := #statInterfaceSignalsHmi[24].valueSymbolRight)
   END_RUNG
   // the same network as SCL:
   #instSignals24Left(signal00 := "BK21"."X10-1.SEPA CLAMP&CUTTER X-AXIS LIMIT SENSOR(-)",   // "LAF_InterfaceSignalsBool"
                      signal01 := "BK21"."X10-2.SEPA CLAMP&CUTTER X-AXIS HOME SENSOR",
                      signal02 := "BK21"."X12-1.SEPA CLAMP&CUTTER X-AXIS LIMIT SENSOR(+)",
                      signal03 := "BK21"."X12-2.SPARE",
                      signal04 := "BK21"."X14-1.SEPA GRIPPER X-AXIS LIMIT SENSOR(-)",
                      signal05 := "BK21"."X14-2.SEPA GRIPPER X-AXIS HOME SENSOR",
                      signal06 := "BK21"."X16-1.SEPA GRIPPER X-AXIS LIMIT SENSOR(+)",
                      signal07 := "BK21"."X16-2.SPARE",
                      interfaceSignals := #statInterfaceSignalsHmi[24].valueSymbolLeft,
                      ENO => #_w1);
   IF #_w1 THEN
       #instSignals24Right(interfaceSignals := #statInterfaceSignalsHmi[24].valueSymbolRight);   // "LAF_InterfaceSignalsBool"
   END_IF;
END_REGION

REGION Network 30: Interface Signals 05 -Example: Model Flex-Pro-Line - IN/OUT- / Interface Signals 25
   // Aufruf des Schnittstellen Signal Bausteins Ba-Bereich 4 / Call the interface signals bool blocks of opmode 4
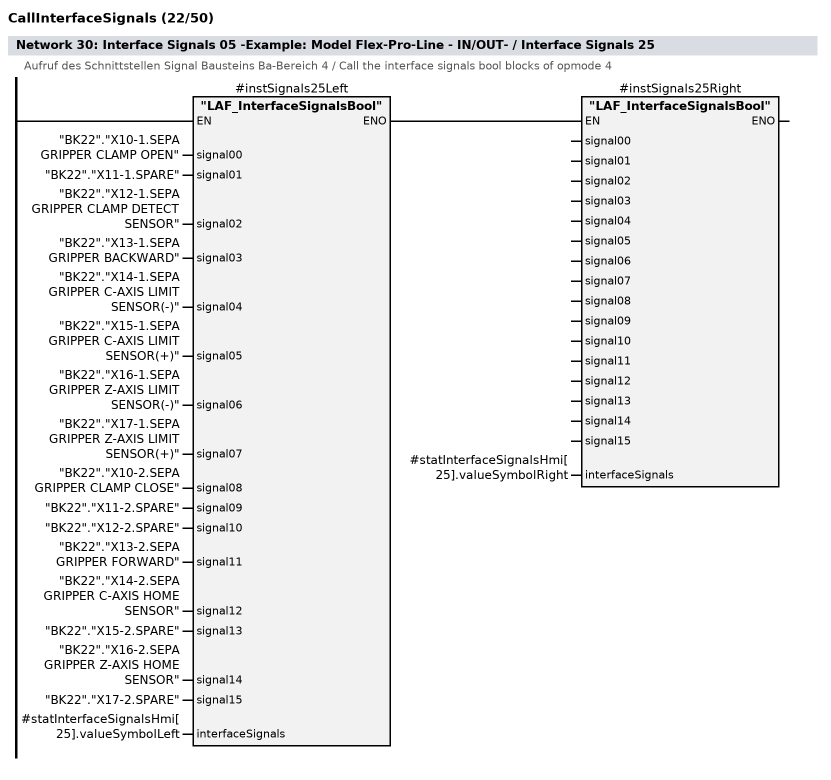
   RUNG wire#powerrail
      #instSignals25Left(signal00 := "BK22"."X10-1.SEPA GRIPPER CLAMP OPEN", signal01 := "BK22"."X11-1.SPARE", signal02 := "BK22"."X12-1.SEPA GRIPPER CLAMP DETECT SENSOR", signal03 := "BK22"."X13-1.SEPA GRIPPER BACKWARD", signal04 := "BK22"."X14-1.SEPA GRIPPER C-AXIS LIMIT SENSOR(-)", signal05 := "BK22"."X15-1.SEPA GRIPPER C-AXIS LIMIT SENSOR(+)", signal06 := "BK22"."X16-1.SEPA GRIPPER Z-AXIS LIMIT SENSOR(-)", signal07 := "BK22"."X17-1.SEPA GRIPPER Z-AXIS LIMIT SENSOR(+)", signal08 := "BK22"."X10-2.SEPA GRIPPER CLAMP CLOSE", signal09 := "BK22"."X11-2.SPARE", signal10 := "BK22"."X12-2.SPARE", signal11 := "BK22"."X13-2.SEPA GRIPPER FORWARD", signal12 := "BK22"."X14-2.SEPA GRIPPER C-AXIS HOME SENSOR", signal13 := "BK22"."X15-2.SPARE", signal14 := "BK22"."X16-2.SEPA GRIPPER Z-AXIS HOME SENSOR", signal15 := "BK22"."X17-2.SPARE", interfaceSignals := #statInterfaceSignalsHmi[25].valueSymbolLeft)
      #instSignals25Right(signal00 :=, signal01 :=, signal02 :=, signal03 :=, signal04 :=, signal05 :=, signal06 :=, signal07 :=, signal08 :=, signal09 :=, signal10 :=, signal11 :=, signal12 :=, signal13 :=, signal14 :=, signal15 :=, interfaceSignals := #statInterfaceSignalsHmi[25].valueSymbolRight)
   END_RUNG
   // the same network as SCL:
   #instSignals25Left(signal00 := "BK22"."X10-1.SEPA GRIPPER CLAMP OPEN",   // "LAF_InterfaceSignalsBool"
                      signal01 := "BK22"."X11-1.SPARE",
                      signal02 := "BK22"."X12-1.SEPA GRIPPER CLAMP DETECT SENSOR",
                      signal03 := "BK22"."X13-1.SEPA GRIPPER BACKWARD",
                      signal04 := "BK22"."X14-1.SEPA GRIPPER C-AXIS LIMIT SENSOR(-)",
                      signal05 := "BK22"."X15-1.SEPA GRIPPER C-AXIS LIMIT SENSOR(+)",
                      signal06 := "BK22"."X16-1.SEPA GRIPPER Z-AXIS LIMIT SENSOR(-)",
                      signal07 := "BK22"."X17-1.SEPA GRIPPER Z-AXIS LIMIT SENSOR(+)",
                      signal08 := "BK22"."X10-2.SEPA GRIPPER CLAMP CLOSE",
                      signal09 := "BK22"."X11-2.SPARE",
                      signal10 := "BK22"."X12-2.SPARE",
                      signal11 := "BK22"."X13-2.SEPA GRIPPER FORWARD",
                      signal12 := "BK22"."X14-2.SEPA GRIPPER C-AXIS HOME SENSOR",
                      signal13 := "BK22"."X15-2.SPARE",
                      signal14 := "BK22"."X16-2.SEPA GRIPPER Z-AXIS HOME SENSOR",
                      signal15 := "BK22"."X17-2.SPARE",
                      interfaceSignals := #statInterfaceSignalsHmi[25].valueSymbolLeft,
                      ENO => #_w1);
   IF #_w1 THEN
       #instSignals25Right(interfaceSignals := #statInterfaceSignalsHmi[25].valueSymbolRight);   // "LAF_InterfaceSignalsBool"
   END_IF;
END_REGION

REGION Network 31: Interface Signals 05 -Example: Model Flex-Pro-Line - IN/OUT- / Interface Signals 26
   // Aufruf des Schnittstellen Signal Bausteins Ba-Bereich 4 / Call the interface signals bool blocks of opmode 4
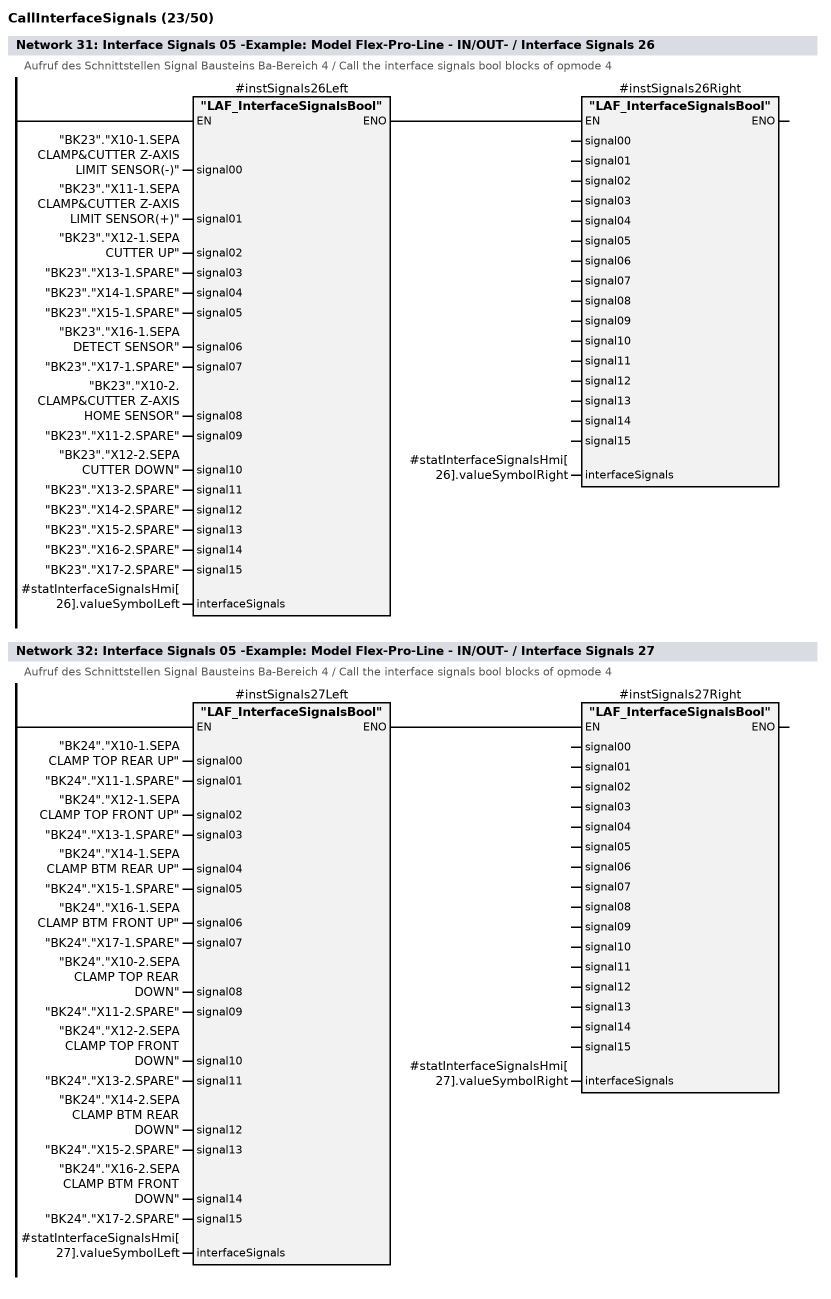
   RUNG wire#powerrail
      #instSignals26Left(signal00 := "BK23"."X10-1.SEPA CLAMP&CUTTER Z-AXIS LIMIT SENSOR(-)", signal01 := "BK23"."X11-1.SEPA CLAMP&CUTTER Z-AXIS LIMIT SENSOR(+)", signal02 := "BK23"."X12-1.SEPA CUTTER UP", signal03 := "BK23"."X13-1.SPARE", signal04 := "BK23"."X14-1.SPARE", signal05 := "BK23"."X15-1.SPARE", signal06 := "BK23"."X16-1.SEPA DETECT SENSOR", signal07 := "BK23"."X17-1.SPARE", signal08 := "BK23"."X10-2.CLAMP&CUTTER Z-AXIS HOME SENSOR", signal09 := "BK23"."X11-2.SPARE", signal10 := "BK23"."X12-2.SEPA CUTTER DOWN", signal11 := "BK23"."X13-2.SPARE", signal12 := "BK23"."X14-2.SPARE", signal13 := "BK23"."X15-2.SPARE", signal14 := "BK23"."X16-2.SPARE", signal15 := "BK23"."X17-2.SPARE", interfaceSignals := #statInterfaceSignalsHmi[26].valueSymbolLeft)
      #instSignals26Right(signal00 :=, signal01 :=, signal02 :=, signal03 :=, signal04 :=, signal05 :=, signal06 :=, signal07 :=, signal08 :=, signal09 :=, signal10 :=, signal11 :=, signal12 :=, signal13 :=, signal14 :=, signal15 :=, interfaceSignals := #statInterfaceSignalsHmi[26].valueSymbolRight)
   END_RUNG
   // the same network as SCL:
   #instSignals26Left(signal00 := "BK23"."X10-1.SEPA CLAMP&CUTTER Z-AXIS LIMIT SENSOR(-)",   // "LAF_InterfaceSignalsBool"
                      signal01 := "BK23"."X11-1.SEPA CLAMP&CUTTER Z-AXIS LIMIT SENSOR(+)",
                      signal02 := "BK23"."X12-1.SEPA CUTTER UP",
                      signal03 := "BK23"."X13-1.SPARE",
                      signal04 := "BK23"."X14-1.SPARE",
                      signal05 := "BK23"."X15-1.SPARE",
                      signal06 := "BK23"."X16-1.SEPA DETECT SENSOR",
                      signal07 := "BK23"."X17-1.SPARE",
                      signal08 := "BK23"."X10-2.CLAMP&CUTTER Z-AXIS HOME SENSOR",
                      signal09 := "BK23"."X11-2.SPARE",
                      signal10 := "BK23"."X12-2.SEPA CUTTER DOWN",
                      signal11 := "BK23"."X13-2.SPARE",
                      signal12 := "BK23"."X14-2.SPARE",
                      signal13 := "BK23"."X15-2.SPARE",
                      signal14 := "BK23"."X16-2.SPARE",
                      signal15 := "BK23"."X17-2.SPARE",
                      interfaceSignals := #statInterfaceSignalsHmi[26].valueSymbolLeft,
                      ENO => #_w1);
   IF #_w1 THEN
       #instSignals26Right(interfaceSignals := #statInterfaceSignalsHmi[26].valueSymbolRight);   // "LAF_InterfaceSignalsBool"
   END_IF;
END_REGION

REGION Network 32: Interface Signals 05 -Example: Model Flex-Pro-Line - IN/OUT- / Interface Signals 27
   // Aufruf des Schnittstellen Signal Bausteins Ba-Bereich 4 / Call the interface signals bool blocks of opmode 4
   RUNG wire#powerrail
      #instSignals27Left(signal00 := "BK24"."X10-1.SEPA CLAMP TOP REAR UP", signal01 := "BK24"."X11-1.SPARE", signal02 := "BK24"."X12-1.SEPA CLAMP TOP FRONT UP", signal03 := "BK24"."X13-1.SPARE", signal04 := "BK24"."X14-1.SEPA CLAMP BTM REAR UP", signal05 := "BK24"."X15-1.SPARE", signal06 := "BK24"."X16-1.SEPA CLAMP BTM FRONT UP", signal07 := "BK24"."X17-1.SPARE", signal08 := "BK24"."X10-2.SEPA CLAMP TOP REAR DOWN", signal09 := "BK24"."X11-2.SPARE", signal10 := "BK24"."X12-2.SEPA CLAMP TOP FRONT DOWN", signal11 := "BK24"."X13-2.SPARE", signal12 := "BK24"."X14-2.SEPA CLAMP BTM REAR DOWN", signal13 := "BK24"."X15-2.SPARE", signal14 := "BK24"."X16-2.SEPA CLAMP BTM FRONT DOWN", signal15 := "BK24"."X17-2.SPARE", interfaceSignals := #statInterfaceSignalsHmi[27].valueSymbolLeft)
      #instSignals27Right(signal00 :=, signal01 :=, signal02 :=, signal03 :=, signal04 :=, signal05 :=, signal06 :=, signal07 :=, signal08 :=, signal09 :=, signal10 :=, signal11 :=, signal12 :=, signal13 :=, signal14 :=, signal15 :=, interfaceSignals := #statInterfaceSignalsHmi[27].valueSymbolRight)
   END_RUNG
   // the same network as SCL:
   #instSignals27Left(signal00 := "BK24"."X10-1.SEPA CLAMP TOP REAR UP",   // "LAF_InterfaceSignalsBool"
                      signal01 := "BK24"."X11-1.SPARE",
                      signal02 := "BK24"."X12-1.SEPA CLAMP TOP FRONT UP",
                      signal03 := "BK24"."X13-1.SPARE",
                      signal04 := "BK24"."X14-1.SEPA CLAMP BTM REAR UP",
                      signal05 := "BK24"."X15-1.SPARE",
                      signal06 := "BK24"."X16-1.SEPA CLAMP BTM FRONT UP",
                      signal07 := "BK24"."X17-1.SPARE",
                      signal08 := "BK24"."X10-2.SEPA CLAMP TOP REAR DOWN",
                      signal09 := "BK24"."X11-2.SPARE",
                      signal10 := "BK24"."X12-2.SEPA CLAMP TOP FRONT DOWN",
                      signal11 := "BK24"."X13-2.SPARE",
                      signal12 := "BK24"."X14-2.SEPA CLAMP BTM REAR DOWN",
                      signal13 := "BK24"."X15-2.SPARE",
                      signal14 := "BK24"."X16-2.SEPA CLAMP BTM FRONT DOWN",
                      signal15 := "BK24"."X17-2.SPARE",
                      interfaceSignals := #statInterfaceSignalsHmi[27].valueSymbolLeft,
                      ENO => #_w1);
   IF #_w1 THEN
       #instSignals27Right(interfaceSignals := #statInterfaceSignalsHmi[27].valueSymbolRight);   // "LAF_InterfaceSignalsBool"
   END_IF;
END_REGION

REGION Network 33: Interface Signals 05 -Example: Model Flex-Pro-Line - IN/OUT- / Interface Signals 28
   // Aufruf des Schnittstellen Signal Bausteins Ba-Bereich 4 / Call the interface signals bool blocks of opmode 4
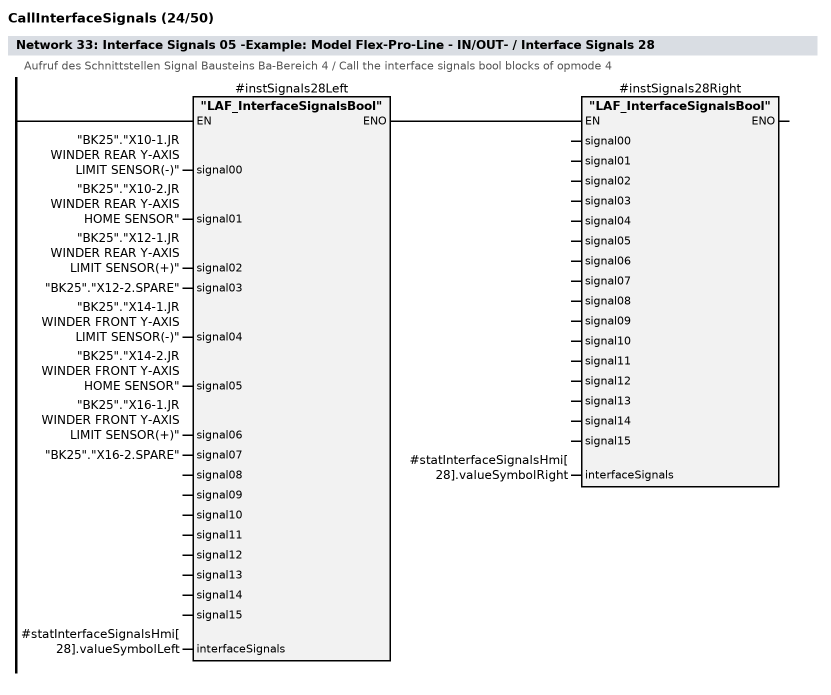
   RUNG wire#powerrail
      #instSignals28Left(signal00 := "BK25"."X10-1.JR WINDER REAR Y-AXIS LIMIT SENSOR(-)", signal01 := "BK25"."X10-2.JR WINDER REAR Y-AXIS HOME SENSOR", signal02 := "BK25"."X12-1.JR WINDER REAR Y-AXIS LIMIT SENSOR(+)", signal03 := "BK25"."X12-2.SPARE", signal04 := "BK25"."X14-1.JR WINDER FRONT Y-AXIS LIMIT SENSOR(-)", signal05 := "BK25"."X14-2.JR WINDER FRONT Y-AXIS HOME SENSOR", signal06 := "BK25"."X16-1.JR WINDER FRONT Y-AXIS LIMIT SENSOR(+)", signal07 := "BK25"."X16-2.SPARE", signal08 :=, signal09 :=, signal10 :=, signal11 :=, signal12 :=, signal13 :=, signal14 :=, signal15 :=, interfaceSignals := #statInterfaceSignalsHmi[28].valueSymbolLeft)
      #instSignals28Right(signal00 :=, signal01 :=, signal02 :=, signal03 :=, signal04 :=, signal05 :=, signal06 :=, signal07 :=, signal08 :=, signal09 :=, signal10 :=, signal11 :=, signal12 :=, signal13 :=, signal14 :=, signal15 :=, interfaceSignals := #statInterfaceSignalsHmi[28].valueSymbolRight)
   END_RUNG
   // the same network as SCL:
   #instSignals28Left(signal00 := "BK25"."X10-1.JR WINDER REAR Y-AXIS LIMIT SENSOR(-)",   // "LAF_InterfaceSignalsBool"
                      signal01 := "BK25"."X10-2.JR WINDER REAR Y-AXIS HOME SENSOR",
                      signal02 := "BK25"."X12-1.JR WINDER REAR Y-AXIS LIMIT SENSOR(+)",
                      signal03 := "BK25"."X12-2.SPARE",
                      signal04 := "BK25"."X14-1.JR WINDER FRONT Y-AXIS LIMIT SENSOR(-)",
                      signal05 := "BK25"."X14-2.JR WINDER FRONT Y-AXIS HOME SENSOR",
                      signal06 := "BK25"."X16-1.JR WINDER FRONT Y-AXIS LIMIT SENSOR(+)",
                      signal07 := "BK25"."X16-2.SPARE",
                      interfaceSignals := #statInterfaceSignalsHmi[28].valueSymbolLeft,
                      ENO => #_w1);
   IF #_w1 THEN
       #instSignals28Right(interfaceSignals := #statInterfaceSignalsHmi[28].valueSymbolRight);   // "LAF_InterfaceSignalsBool"
   END_IF;
END_REGION

REGION Network 34: Interface Signals 05 -Example: Model Flex-Pro-Line - IN/OUT- / Interface Signals 29
   // Aufruf des Schnittstellen Signal Bausteins Ba-Bereich 4 / Call the interface signals bool blocks of opmode 4
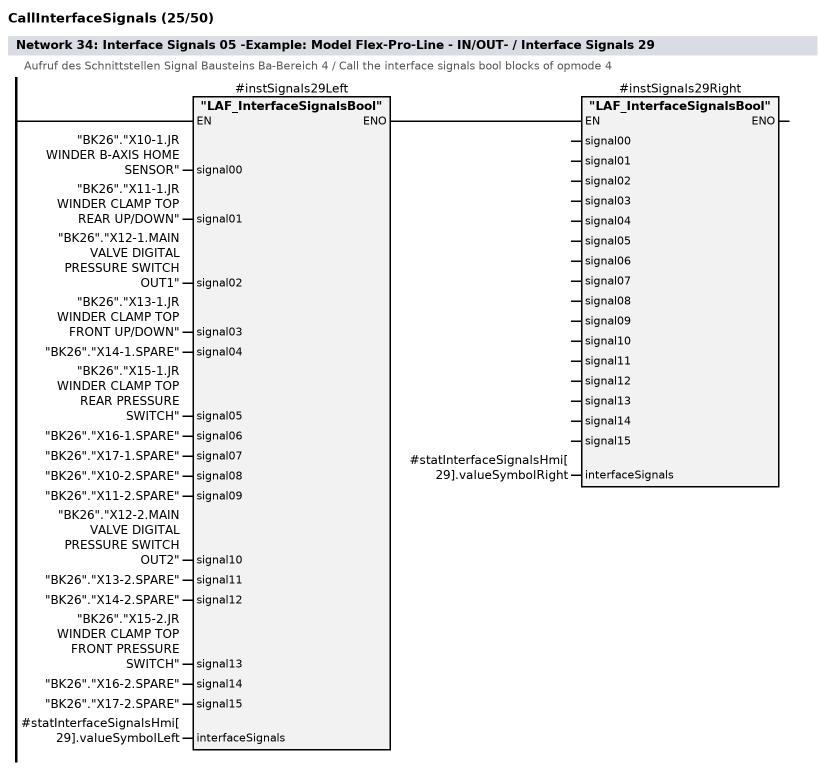
   RUNG wire#powerrail
      #instSignals29Left(signal00 := "BK26"."X10-1.JR WINDER B-AXIS HOME SENSOR", signal01 := "BK26"."X11-1.JR WINDER CLAMP TOP REAR UP/DOWN", signal02 := "BK26"."X12-1.MAIN VALVE DIGITAL PRESSURE SWITCH OUT1", signal03 := "BK26"."X13-1.JR WINDER CLAMP TOP FRONT UP/DOWN", signal04 := "BK26"."X14-1.SPARE", signal05 := "BK26"."X15-1.JR WINDER CLAMP TOP REAR PRESSURE SWITCH", signal06 := "BK26"."X16-1.SPARE", signal07 := "BK26"."X17-1.SPARE", signal08 := "BK26"."X10-2.SPARE", signal09 := "BK26"."X11-2.SPARE", signal10 := "BK26"."X12-2.MAIN VALVE DIGITAL PRESSURE SWITCH OUT2", signal11 := "BK26"."X13-2.SPARE", signal12 := "BK26"."X14-2.SPARE", signal13 := "BK26"."X15-2.JR WINDER CLAMP TOP FRONT PRESSURE SWITCH", signal14 := "BK26"."X16-2.SPARE", signal15 := "BK26"."X17-2.SPARE", interfaceSignals := #statInterfaceSignalsHmi[29].valueSymbolLeft)
      #instSignals29Right(signal00 :=, signal01 :=, signal02 :=, signal03 :=, signal04 :=, signal05 :=, signal06 :=, signal07 :=, signal08 :=, signal09 :=, signal10 :=, signal11 :=, signal12 :=, signal13 :=, signal14 :=, signal15 :=, interfaceSignals := #statInterfaceSignalsHmi[29].valueSymbolRight)
   END_RUNG
   // the same network as SCL:
   #instSignals29Left(signal00 := "BK26"."X10-1.JR WINDER B-AXIS HOME SENSOR",   // "LAF_InterfaceSignalsBool"
                      signal01 := "BK26"."X11-1.JR WINDER CLAMP TOP REAR UP/DOWN",
                      signal02 := "BK26"."X12-1.MAIN VALVE DIGITAL PRESSURE SWITCH OUT1",
                      signal03 := "BK26"."X13-1.JR WINDER CLAMP TOP FRONT UP/DOWN",
                      signal04 := "BK26"."X14-1.SPARE",
                      signal05 := "BK26"."X15-1.JR WINDER CLAMP TOP REAR PRESSURE SWITCH",
                      signal06 := "BK26"."X16-1.SPARE",
                      signal07 := "BK26"."X17-1.SPARE",
                      signal08 := "BK26"."X10-2.SPARE",
                      signal09 := "BK26"."X11-2.SPARE",
                      signal10 := "BK26"."X12-2.MAIN VALVE DIGITAL PRESSURE SWITCH OUT2",
                      signal11 := "BK26"."X13-2.SPARE",
                      signal12 := "BK26"."X14-2.SPARE",
                      signal13 := "BK26"."X15-2.JR WINDER CLAMP TOP FRONT PRESSURE SWITCH",
                      signal14 := "BK26"."X16-2.SPARE",
                      signal15 := "BK26"."X17-2.SPARE",
                      interfaceSignals := #statInterfaceSignalsHmi[29].valueSymbolLeft,
                      ENO => #_w1);
   IF #_w1 THEN
       #instSignals29Right(interfaceSignals := #statInterfaceSignalsHmi[29].valueSymbolRight);   // "LAF_InterfaceSignalsBool"
   END_IF;
END_REGION

REGION Network 35: Interface Signals 05 -Example: Model Flex-Pro-Line - IN/OUT- / Interface Signals 30
   // Aufruf des Schnittstellen Signal Bausteins Ba-Bereich 4 / Call the interface signals bool blocks of opmode 4
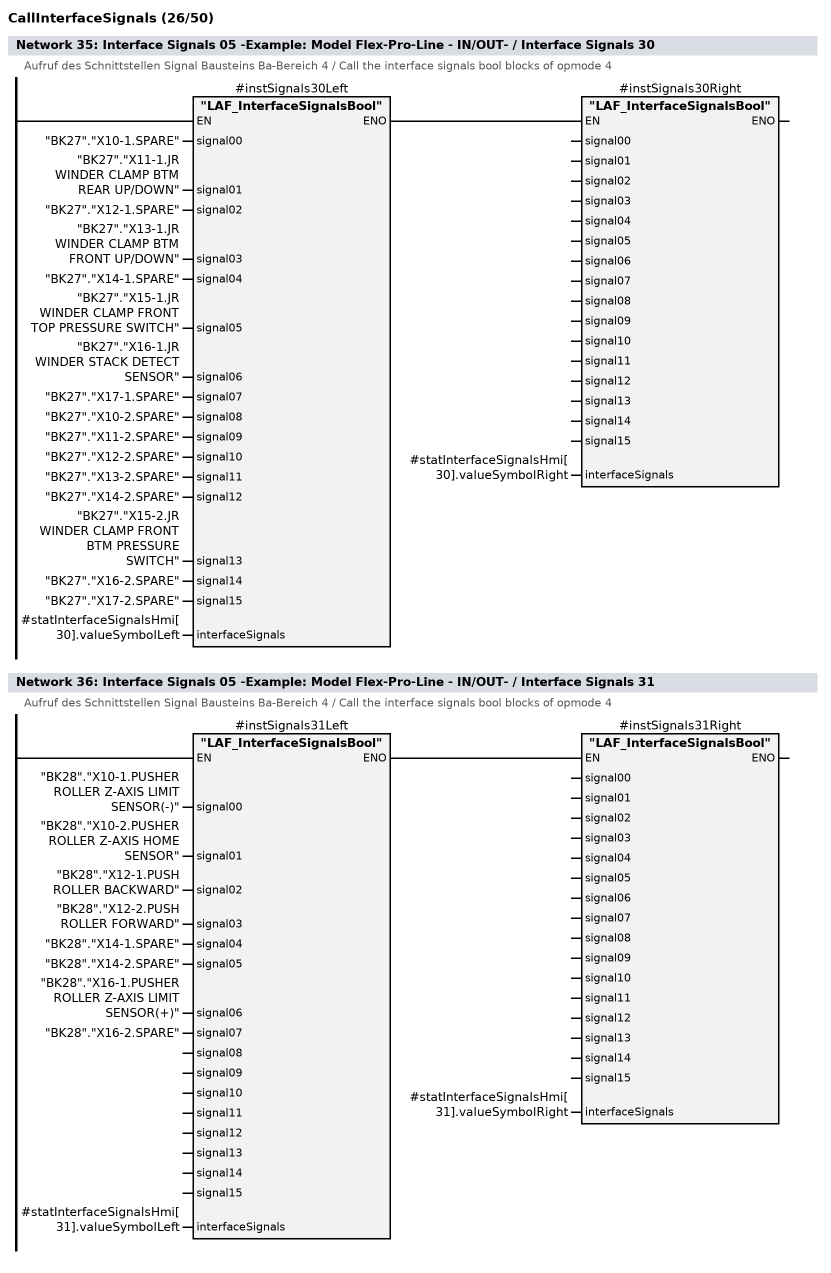
   RUNG wire#powerrail
      #instSignals30Left(signal00 := "BK27"."X10-1.SPARE", signal01 := "BK27"."X11-1.JR WINDER CLAMP BTM REAR UP/DOWN", signal02 := "BK27"."X12-1.SPARE", signal03 := "BK27"."X13-1.JR WINDER CLAMP BTM FRONT UP/DOWN", signal04 := "BK27"."X14-1.SPARE", signal05 := "BK27"."X15-1.JR WINDER CLAMP FRONT TOP PRESSURE SWITCH", signal06 := "BK27"."X16-1.JR WINDER STACK DETECT SENSOR", signal07 := "BK27"."X17-1.SPARE", signal08 := "BK27"."X10-2.SPARE", signal09 := "BK27"."X11-2.SPARE", signal10 := "BK27"."X12-2.SPARE", signal11 := "BK27"."X13-2.SPARE", signal12 := "BK27"."X14-2.SPARE", signal13 := "BK27"."X15-2.JR WINDER CLAMP FRONT BTM PRESSURE SWITCH", signal14 := "BK27"."X16-2.SPARE", signal15 := "BK27"."X17-2.SPARE", interfaceSignals := #statInterfaceSignalsHmi[30].valueSymbolLeft)
      #instSignals30Right(signal00 :=, signal01 :=, signal02 :=, signal03 :=, signal04 :=, signal05 :=, signal06 :=, signal07 :=, signal08 :=, signal09 :=, signal10 :=, signal11 :=, signal12 :=, signal13 :=, signal14 :=, signal15 :=, interfaceSignals := #statInterfaceSignalsHmi[30].valueSymbolRight)
   END_RUNG
   // the same network as SCL:
   #instSignals30Left(signal00 := "BK27"."X10-1.SPARE",   // "LAF_InterfaceSignalsBool"
                      signal01 := "BK27"."X11-1.JR WINDER CLAMP BTM REAR UP/DOWN",
                      signal02 := "BK27"."X12-1.SPARE",
                      signal03 := "BK27"."X13-1.JR WINDER CLAMP BTM FRONT UP/DOWN",
                      signal04 := "BK27"."X14-1.SPARE",
                      signal05 := "BK27"."X15-1.JR WINDER CLAMP FRONT TOP PRESSURE SWITCH",
                      signal06 := "BK27"."X16-1.JR WINDER STACK DETECT SENSOR",
                      signal07 := "BK27"."X17-1.SPARE",
                      signal08 := "BK27"."X10-2.SPARE",
                      signal09 := "BK27"."X11-2.SPARE",
                      signal10 := "BK27"."X12-2.SPARE",
                      signal11 := "BK27"."X13-2.SPARE",
                      signal12 := "BK27"."X14-2.SPARE",
                      signal13 := "BK27"."X15-2.JR WINDER CLAMP FRONT BTM PRESSURE SWITCH",
                      signal14 := "BK27"."X16-2.SPARE",
                      signal15 := "BK27"."X17-2.SPARE",
                      interfaceSignals := #statInterfaceSignalsHmi[30].valueSymbolLeft,
                      ENO => #_w1);
   IF #_w1 THEN
       #instSignals30Right(interfaceSignals := #statInterfaceSignalsHmi[30].valueSymbolRight);   // "LAF_InterfaceSignalsBool"
   END_IF;
END_REGION

REGION Network 36: Interface Signals 05 -Example: Model Flex-Pro-Line - IN/OUT- / Interface Signals 31
   // Aufruf des Schnittstellen Signal Bausteins Ba-Bereich 4 / Call the interface signals bool blocks of opmode 4
   RUNG wire#powerrail
      #instSignals31Left(signal00 := "BK28"."X10-1.PUSHER ROLLER Z-AXIS LIMIT SENSOR(-)", signal01 := "BK28"."X10-2.PUSHER ROLLER Z-AXIS HOME SENSOR", signal02 := "BK28"."X12-1.PUSH ROLLER BACKWARD", signal03 := "BK28"."X12-2.PUSH ROLLER FORWARD", signal04 := "BK28"."X14-1.SPARE", signal05 := "BK28"."X14-2.SPARE", signal06 := "BK28"."X16-1.PUSHER ROLLER Z-AXIS LIMIT SENSOR(+)", signal07 := "BK28"."X16-2.SPARE", signal08 :=, signal09 :=, signal10 :=, signal11 :=, signal12 :=, signal13 :=, signal14 :=, signal15 :=, interfaceSignals := #statInterfaceSignalsHmi[31].valueSymbolLeft)
      #instSignals31Right(signal00 :=, signal01 :=, signal02 :=, signal03 :=, signal04 :=, signal05 :=, signal06 :=, signal07 :=, signal08 :=, signal09 :=, signal10 :=, signal11 :=, signal12 :=, signal13 :=, signal14 :=, signal15 :=, interfaceSignals := #statInterfaceSignalsHmi[31].valueSymbolRight)
   END_RUNG
   // the same network as SCL:
   #instSignals31Left(signal00 := "BK28"."X10-1.PUSHER ROLLER Z-AXIS LIMIT SENSOR(-)",   // "LAF_InterfaceSignalsBool"
                      signal01 := "BK28"."X10-2.PUSHER ROLLER Z-AXIS HOME SENSOR",
                      signal02 := "BK28"."X12-1.PUSH ROLLER BACKWARD",
                      signal03 := "BK28"."X12-2.PUSH ROLLER FORWARD",
                      signal04 := "BK28"."X14-1.SPARE",
                      signal05 := "BK28"."X14-2.SPARE",
                      signal06 := "BK28"."X16-1.PUSHER ROLLER Z-AXIS LIMIT SENSOR(+)",
                      signal07 := "BK28"."X16-2.SPARE",
                      interfaceSignals := #statInterfaceSignalsHmi[31].valueSymbolLeft,
                      ENO => #_w1);
   IF #_w1 THEN
       #instSignals31Right(interfaceSignals := #statInterfaceSignalsHmi[31].valueSymbolRight);   // "LAF_InterfaceSignalsBool"
   END_IF;
END_REGION

REGION Network 37: Interface Signals 05 -Example: Model Flex-Pro-Line - IN/OUT- / Interface Signals 32
   // Aufruf des Schnittstellen Signal Bausteins Ba-Bereich 4 / Call the interface signals bool blocks of opmode 4
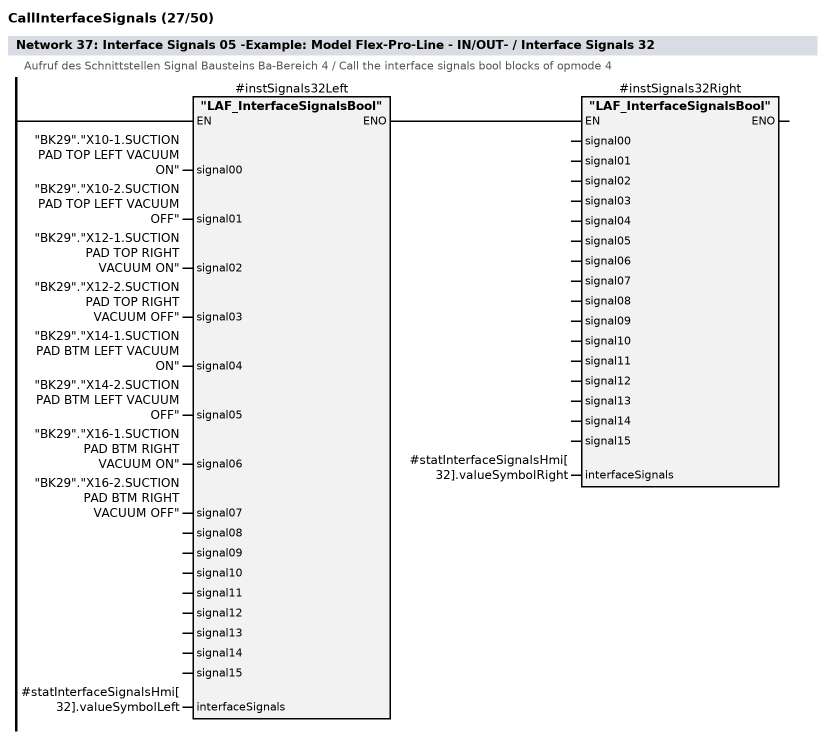
   RUNG wire#powerrail
      #instSignals32Left(signal00 := "BK29"."X10-1.SUCTION PAD TOP LEFT VACUUM ON", signal01 := "BK29"."X10-2.SUCTION PAD TOP LEFT VACUUM OFF", signal02 := "BK29"."X12-1.SUCTION PAD TOP RIGHT VACUUM ON", signal03 := "BK29"."X12-2.SUCTION PAD TOP RIGHT VACUUM OFF", signal04 := "BK29"."X14-1.SUCTION PAD BTM LEFT VACUUM ON", signal05 := "BK29"."X14-2.SUCTION PAD BTM LEFT VACUUM OFF", signal06 := "BK29"."X16-1.SUCTION PAD BTM RIGHT VACUUM ON", signal07 := "BK29"."X16-2.SUCTION PAD BTM RIGHT VACUUM OFF", signal08 :=, signal09 :=, signal10 :=, signal11 :=, signal12 :=, signal13 :=, signal14 :=, signal15 :=, interfaceSignals := #statInterfaceSignalsHmi[32].valueSymbolLeft)
      #instSignals32Right(signal00 :=, signal01 :=, signal02 :=, signal03 :=, signal04 :=, signal05 :=, signal06 :=, signal07 :=, signal08 :=, signal09 :=, signal10 :=, signal11 :=, signal12 :=, signal13 :=, signal14 :=, signal15 :=, interfaceSignals := #statInterfaceSignalsHmi[32].valueSymbolRight)
   END_RUNG
   // the same network as SCL:
   #instSignals32Left(signal00 := "BK29"."X10-1.SUCTION PAD TOP LEFT VACUUM ON",   // "LAF_InterfaceSignalsBool"
                      signal01 := "BK29"."X10-2.SUCTION PAD TOP LEFT VACUUM OFF",
                      signal02 := "BK29"."X12-1.SUCTION PAD TOP RIGHT VACUUM ON",
                      signal03 := "BK29"."X12-2.SUCTION PAD TOP RIGHT VACUUM OFF",
                      signal04 := "BK29"."X14-1.SUCTION PAD BTM LEFT VACUUM ON",
                      signal05 := "BK29"."X14-2.SUCTION PAD BTM LEFT VACUUM OFF",
                      signal06 := "BK29"."X16-1.SUCTION PAD BTM RIGHT VACUUM ON",
                      signal07 := "BK29"."X16-2.SUCTION PAD BTM RIGHT VACUUM OFF",
                      interfaceSignals := #statInterfaceSignalsHmi[32].valueSymbolLeft,
                      ENO => #_w1);
   IF #_w1 THEN
       #instSignals32Right(interfaceSignals := #statInterfaceSignalsHmi[32].valueSymbolRight);   // "LAF_InterfaceSignalsBool"
   END_IF;
END_REGION

REGION Network 38: Interface Signals 03 -Example: System flags & Clock flags- / Interface Signals33
   // Aufruf des Schnittstellen Signal Bausteins für die Systemvariablen / Call the interface signals bool blocks of system tags
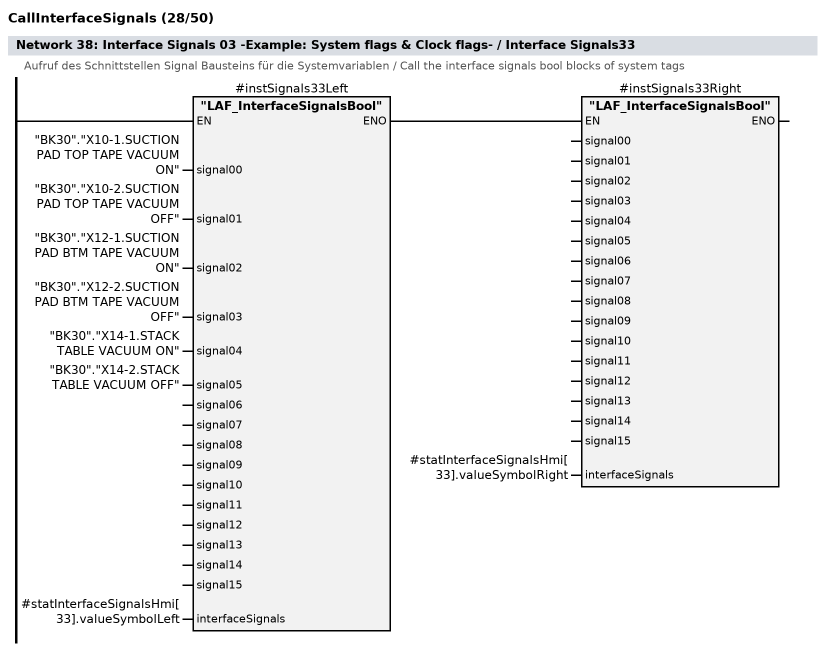
   RUNG wire#powerrail
      #instSignals33Left(signal00 := "BK30"."X10-1.SUCTION PAD TOP TAPE VACUUM ON", signal01 := "BK30"."X10-2.SUCTION PAD TOP TAPE VACUUM OFF", signal02 := "BK30"."X12-1.SUCTION PAD BTM TAPE VACUUM ON", signal03 := "BK30"."X12-2.SUCTION PAD BTM TAPE VACUUM OFF", signal04 := "BK30"."X14-1.STACK TABLE VACUUM ON", signal05 := "BK30"."X14-2.STACK TABLE VACUUM OFF", signal06 :=, signal07 :=, signal08 :=, signal09 :=, signal10 :=, signal11 :=, signal12 :=, signal13 :=, signal14 :=, signal15 :=, interfaceSignals := #statInterfaceSignalsHmi[33].valueSymbolLeft)
      #instSignals33Right(signal00 :=, signal01 :=, signal02 :=, signal03 :=, signal04 :=, signal05 :=, signal06 :=, signal07 :=, signal08 :=, signal09 :=, signal10 :=, signal11 :=, signal12 :=, signal13 :=, signal14 :=, signal15 :=, interfaceSignals := #statInterfaceSignalsHmi[33].valueSymbolRight)
   END_RUNG
   // the same network as SCL:
   #instSignals33Left(signal00 := "BK30"."X10-1.SUCTION PAD TOP TAPE VACUUM ON",   // "LAF_InterfaceSignalsBool"
                      signal01 := "BK30"."X10-2.SUCTION PAD TOP TAPE VACUUM OFF",
                      signal02 := "BK30"."X12-1.SUCTION PAD BTM TAPE VACUUM ON",
                      signal03 := "BK30"."X12-2.SUCTION PAD BTM TAPE VACUUM OFF",
                      signal04 := "BK30"."X14-1.STACK TABLE VACUUM ON",
                      signal05 := "BK30"."X14-2.STACK TABLE VACUUM OFF",
                      interfaceSignals := #statInterfaceSignalsHmi[33].valueSymbolLeft,
                      ENO => #_w1);
   IF #_w1 THEN
       #instSignals33Right(interfaceSignals := #statInterfaceSignalsHmi[33].valueSymbolRight);   // "LAF_InterfaceSignalsBool"
   END_IF;
END_REGION

REGION Network 39: Interface Signals 04 -Example: Model Flex-Pro-Line - IN/OUT- / Interface Signals 34
   // Aufruf des Schnittstellen Signal Bausteins Ba-Bereich 4 / Call the interface signals bool blocks of opmode 4
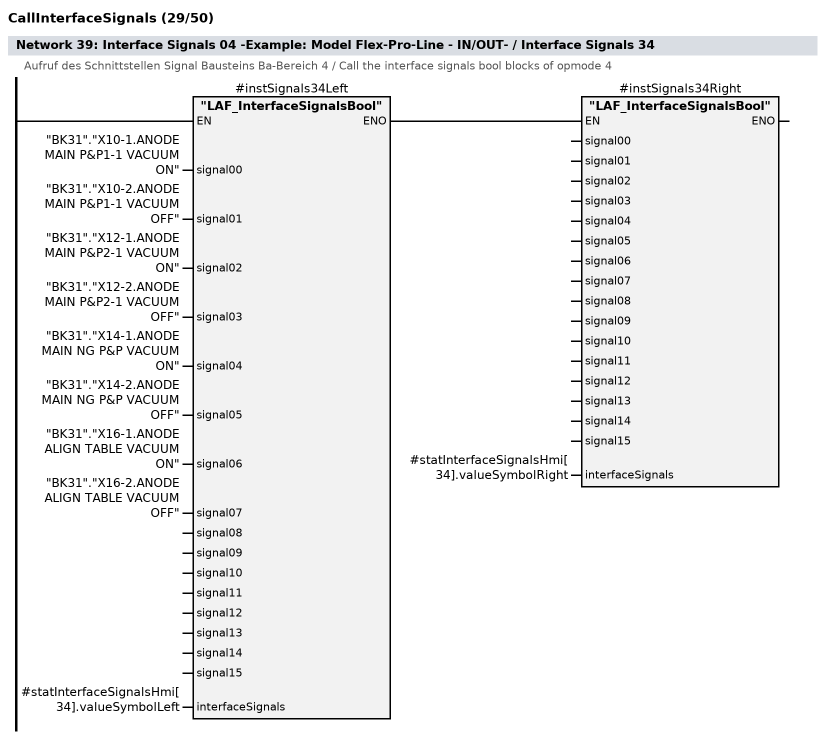
   RUNG wire#powerrail
      #instSignals34Left(signal00 := "BK31"."X10-1.ANODE MAIN P&P1-1 VACUUM ON", signal01 := "BK31"."X10-2.ANODE MAIN P&P1-1 VACUUM OFF", signal02 := "BK31"."X12-1.ANODE MAIN P&P2-1 VACUUM ON", signal03 := "BK31"."X12-2.ANODE MAIN P&P2-1 VACUUM OFF", signal04 := "BK31"."X14-1.ANODE MAIN NG P&P VACUUM ON", signal05 := "BK31"."X14-2.ANODE MAIN NG P&P VACUUM OFF", signal06 := "BK31"."X16-1.ANODE ALIGN TABLE VACUUM ON", signal07 := "BK31"."X16-2.ANODE ALIGN TABLE VACUUM OFF", signal08 :=, signal09 :=, signal10 :=, signal11 :=, signal12 :=, signal13 :=, signal14 :=, signal15 :=, interfaceSignals := #statInterfaceSignalsHmi[34].valueSymbolLeft)
      #instSignals34Right(signal00 :=, signal01 :=, signal02 :=, signal03 :=, signal04 :=, signal05 :=, signal06 :=, signal07 :=, signal08 :=, signal09 :=, signal10 :=, signal11 :=, signal12 :=, signal13 :=, signal14 :=, signal15 :=, interfaceSignals := #statInterfaceSignalsHmi[34].valueSymbolRight)
   END_RUNG
   // the same network as SCL:
   #instSignals34Left(signal00 := "BK31"."X10-1.ANODE MAIN P&P1-1 VACUUM ON",   // "LAF_InterfaceSignalsBool"
                      signal01 := "BK31"."X10-2.ANODE MAIN P&P1-1 VACUUM OFF",
                      signal02 := "BK31"."X12-1.ANODE MAIN P&P2-1 VACUUM ON",
                      signal03 := "BK31"."X12-2.ANODE MAIN P&P2-1 VACUUM OFF",
                      signal04 := "BK31"."X14-1.ANODE MAIN NG P&P VACUUM ON",
                      signal05 := "BK31"."X14-2.ANODE MAIN NG P&P VACUUM OFF",
                      signal06 := "BK31"."X16-1.ANODE ALIGN TABLE VACUUM ON",
                      signal07 := "BK31"."X16-2.ANODE ALIGN TABLE VACUUM OFF",
                      interfaceSignals := #statInterfaceSignalsHmi[34].valueSymbolLeft,
                      ENO => #_w1);
   IF #_w1 THEN
       #instSignals34Right(interfaceSignals := #statInterfaceSignalsHmi[34].valueSymbolRight);   // "LAF_InterfaceSignalsBool"
   END_IF;
END_REGION

REGION Network 40: Interface Signals 05 -Example: Model Flex-Pro-Line - IN/OUT- / Interface Signals 35
   // Aufruf des Schnittstellen Signal Bausteins Ba-Bereich 4 / Call the interface signals bool blocks of opmode 4
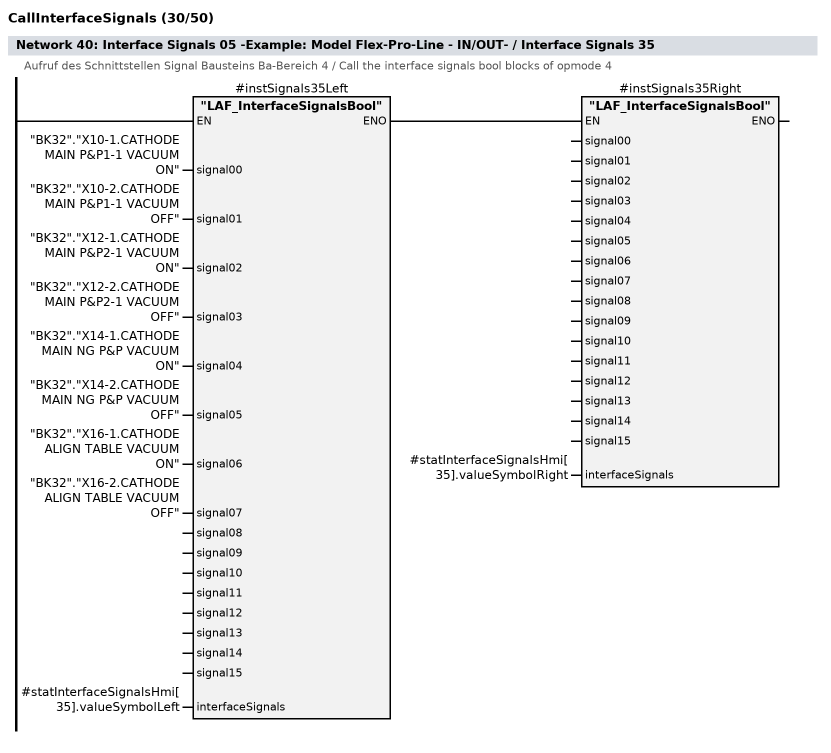
   RUNG wire#powerrail
      #instSignals35Left(signal00 := "BK32"."X10-1.CATHODE MAIN P&P1-1 VACUUM ON", signal01 := "BK32"."X10-2.CATHODE MAIN P&P1-1 VACUUM OFF", signal02 := "BK32"."X12-1.CATHODE MAIN P&P2-1 VACUUM ON", signal03 := "BK32"."X12-2.CATHODE MAIN P&P2-1 VACUUM OFF", signal04 := "BK32"."X14-1.CATHODE MAIN NG P&P VACUUM ON", signal05 := "BK32"."X14-2.CATHODE MAIN NG P&P VACUUM OFF", signal06 := "BK32"."X16-1.CATHODE ALIGN TABLE VACUUM ON", signal07 := "BK32"."X16-2.CATHODE ALIGN TABLE VACUUM OFF", signal08 :=, signal09 :=, signal10 :=, signal11 :=, signal12 :=, signal13 :=, signal14 :=, signal15 :=, interfaceSignals := #statInterfaceSignalsHmi[35].valueSymbolLeft)
      #instSignals35Right(signal00 :=, signal01 :=, signal02 :=, signal03 :=, signal04 :=, signal05 :=, signal06 :=, signal07 :=, signal08 :=, signal09 :=, signal10 :=, signal11 :=, signal12 :=, signal13 :=, signal14 :=, signal15 :=, interfaceSignals := #statInterfaceSignalsHmi[35].valueSymbolRight)
   END_RUNG
   // the same network as SCL:
   #instSignals35Left(signal00 := "BK32"."X10-1.CATHODE MAIN P&P1-1 VACUUM ON",   // "LAF_InterfaceSignalsBool"
                      signal01 := "BK32"."X10-2.CATHODE MAIN P&P1-1 VACUUM OFF",
                      signal02 := "BK32"."X12-1.CATHODE MAIN P&P2-1 VACUUM ON",
                      signal03 := "BK32"."X12-2.CATHODE MAIN P&P2-1 VACUUM OFF",
                      signal04 := "BK32"."X14-1.CATHODE MAIN NG P&P VACUUM ON",
                      signal05 := "BK32"."X14-2.CATHODE MAIN NG P&P VACUUM OFF",
                      signal06 := "BK32"."X16-1.CATHODE ALIGN TABLE VACUUM ON",
                      signal07 := "BK32"."X16-2.CATHODE ALIGN TABLE VACUUM OFF",
                      interfaceSignals := #statInterfaceSignalsHmi[35].valueSymbolLeft,
                      ENO => #_w1);
   IF #_w1 THEN
       #instSignals35Right(interfaceSignals := #statInterfaceSignalsHmi[35].valueSymbolRight);   // "LAF_InterfaceSignalsBool"
   END_IF;
END_REGION

REGION Network 41: Interface Signals 05 -Example: Model Flex-Pro-Line - IN/OUT- / Interface Signals 36
   // Aufruf des Schnittstellen Signal Bausteins Ba-Bereich 4 / Call the interface signals bool blocks of opmode 4
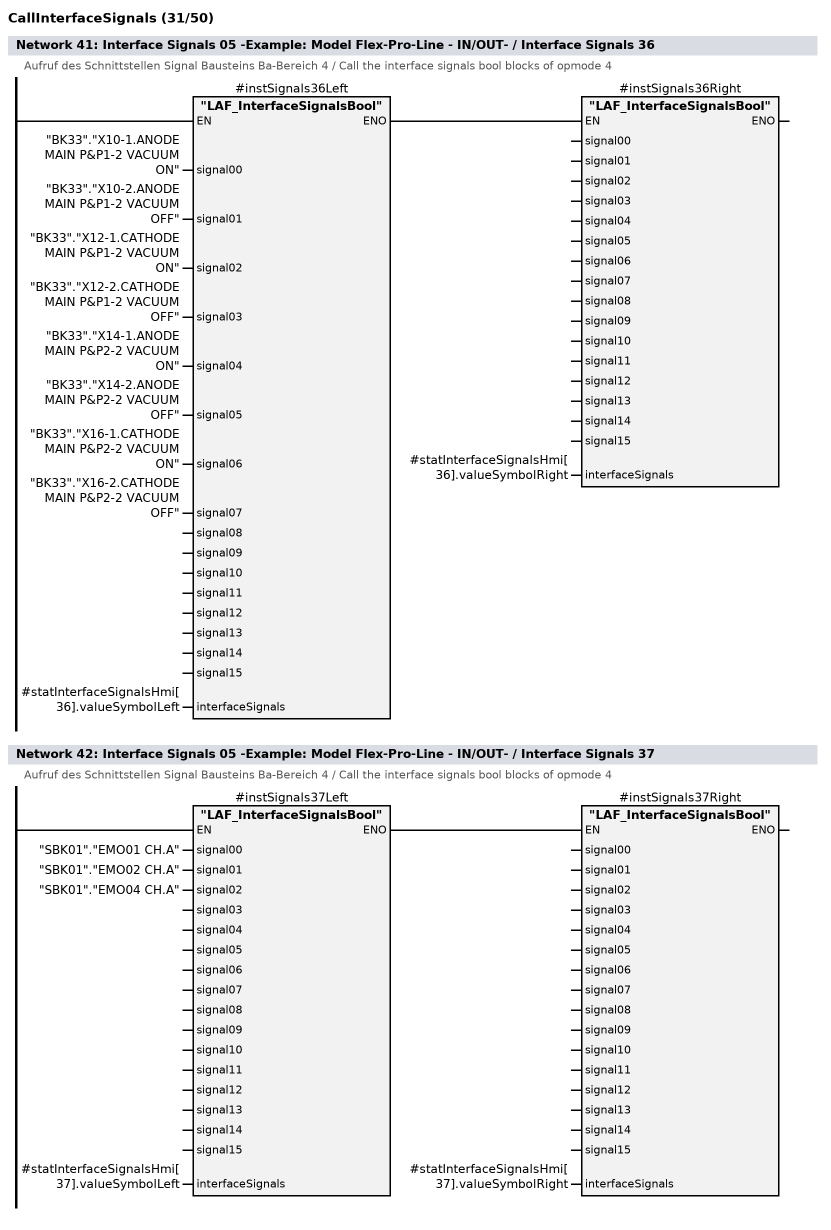
   RUNG wire#powerrail
      #instSignals36Left(signal00 := "BK33"."X10-1.ANODE MAIN P&P1-2 VACUUM ON", signal01 := "BK33"."X10-2.ANODE MAIN P&P1-2 VACUUM OFF", signal02 := "BK33"."X12-1.CATHODE MAIN P&P1-2 VACUUM ON", signal03 := "BK33"."X12-2.CATHODE MAIN P&P1-2 VACUUM OFF", signal04 := "BK33"."X14-1.ANODE MAIN P&P2-2 VACUUM ON", signal05 := "BK33"."X14-2.ANODE MAIN P&P2-2 VACUUM OFF", signal06 := "BK33"."X16-1.CATHODE MAIN P&P2-2 VACUUM ON", signal07 := "BK33"."X16-2.CATHODE MAIN P&P2-2 VACUUM OFF", signal08 :=, signal09 :=, signal10 :=, signal11 :=, signal12 :=, signal13 :=, signal14 :=, signal15 :=, interfaceSignals := #statInterfaceSignalsHmi[36].valueSymbolLeft)
      #instSignals36Right(signal00 :=, signal01 :=, signal02 :=, signal03 :=, signal04 :=, signal05 :=, signal06 :=, signal07 :=, signal08 :=, signal09 :=, signal10 :=, signal11 :=, signal12 :=, signal13 :=, signal14 :=, signal15 :=, interfaceSignals := #statInterfaceSignalsHmi[36].valueSymbolRight)
   END_RUNG
   // the same network as SCL:
   #instSignals36Left(signal00 := "BK33"."X10-1.ANODE MAIN P&P1-2 VACUUM ON",   // "LAF_InterfaceSignalsBool"
                      signal01 := "BK33"."X10-2.ANODE MAIN P&P1-2 VACUUM OFF",
                      signal02 := "BK33"."X12-1.CATHODE MAIN P&P1-2 VACUUM ON",
                      signal03 := "BK33"."X12-2.CATHODE MAIN P&P1-2 VACUUM OFF",
                      signal04 := "BK33"."X14-1.ANODE MAIN P&P2-2 VACUUM ON",
                      signal05 := "BK33"."X14-2.ANODE MAIN P&P2-2 VACUUM OFF",
                      signal06 := "BK33"."X16-1.CATHODE MAIN P&P2-2 VACUUM ON",
                      signal07 := "BK33"."X16-2.CATHODE MAIN P&P2-2 VACUUM OFF",
                      interfaceSignals := #statInterfaceSignalsHmi[36].valueSymbolLeft,
                      ENO => #_w1);
   IF #_w1 THEN
       #instSignals36Right(interfaceSignals := #statInterfaceSignalsHmi[36].valueSymbolRight);   // "LAF_InterfaceSignalsBool"
   END_IF;
END_REGION

REGION Network 42: Interface Signals 05 -Example: Model Flex-Pro-Line - IN/OUT- / Interface Signals 37
   // Aufruf des Schnittstellen Signal Bausteins Ba-Bereich 4 / Call the interface signals bool blocks of opmode 4
   RUNG wire#powerrail
      #instSignals37Left(signal00 := "SBK01"."EMO01 CH.A", signal01 := "SBK01"."EMO02 CH.A", signal02 := "SBK01"."EMO04 CH.A", signal03 :=, signal04 :=, signal05 :=, signal06 :=, signal07 :=, signal08 :=, signal09 :=, signal10 :=, signal11 :=, signal12 :=, signal13 :=, signal14 :=, signal15 :=, interfaceSignals := #statInterfaceSignalsHmi[37].valueSymbolLeft)
      #instSignals37Right(signal00 :=, signal01 :=, signal02 :=, signal03 :=, signal04 :=, signal05 :=, signal06 :=, signal07 :=, signal08 :=, signal09 :=, signal10 :=, signal11 :=, signal12 :=, signal13 :=, signal14 :=, signal15 :=, interfaceSignals := #statInterfaceSignalsHmi[37].valueSymbolRight)
   END_RUNG
   // the same network as SCL:
   #instSignals37Left(signal00 := "SBK01"."EMO01 CH.A",   // "LAF_InterfaceSignalsBool"
                      signal01 := "SBK01"."EMO02 CH.A",
                      signal02 := "SBK01"."EMO04 CH.A",
                      interfaceSignals := #statInterfaceSignalsHmi[37].valueSymbolLeft,
                      ENO => #_w1);
   IF #_w1 THEN
       #instSignals37Right(interfaceSignals := #statInterfaceSignalsHmi[37].valueSymbolRight);   // "LAF_InterfaceSignalsBool"
   END_IF;
END_REGION

REGION Network 43: Interface Signals 05 -Example: Model Flex-Pro-Line - IN/OUT- / Interface Signals 38
   // Aufruf des Schnittstellen Signal Bausteins Ba-Bereich 4 / Call the interface signals bool blocks of opmode 4
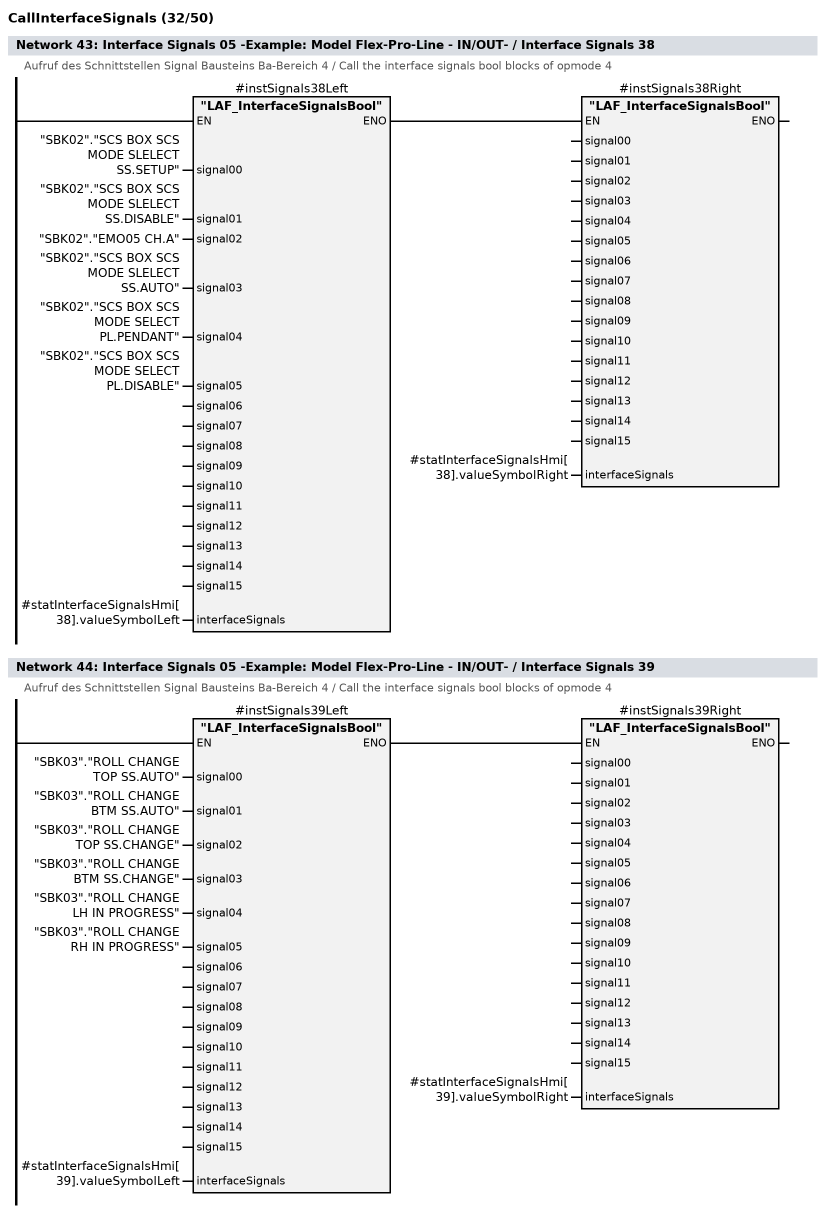
   RUNG wire#powerrail
      #instSignals38Left(signal00 := "SBK02"."SCS BOX SCS MODE SLELECT SS.SETUP", signal01 := "SBK02"."SCS BOX SCS MODE SLELECT SS.DISABLE", signal02 := "SBK02"."EMO05 CH.A", signal03 := "SBK02"."SCS BOX SCS MODE SLELECT SS.AUTO", signal04 := "SBK02"."SCS BOX SCS MODE SELECT PL.PENDANT", signal05 := "SBK02"."SCS BOX SCS MODE SELECT PL.DISABLE", signal06 :=, signal07 :=, signal08 :=, signal09 :=, signal10 :=, signal11 :=, signal12 :=, signal13 :=, signal14 :=, signal15 :=, interfaceSignals := #statInterfaceSignalsHmi[38].valueSymbolLeft)
      #instSignals38Right(signal00 :=, signal01 :=, signal02 :=, signal03 :=, signal04 :=, signal05 :=, signal06 :=, signal07 :=, signal08 :=, signal09 :=, signal10 :=, signal11 :=, signal12 :=, signal13 :=, signal14 :=, signal15 :=, interfaceSignals := #statInterfaceSignalsHmi[38].valueSymbolRight)
   END_RUNG
   // the same network as SCL:
   #instSignals38Left(signal00 := "SBK02"."SCS BOX SCS MODE SLELECT SS.SETUP",   // "LAF_InterfaceSignalsBool"
                      signal01 := "SBK02"."SCS BOX SCS MODE SLELECT SS.DISABLE",
                      signal02 := "SBK02"."EMO05 CH.A",
                      signal03 := "SBK02"."SCS BOX SCS MODE SLELECT SS.AUTO",
                      signal04 := "SBK02"."SCS BOX SCS MODE SELECT PL.PENDANT",
                      signal05 := "SBK02"."SCS BOX SCS MODE SELECT PL.DISABLE",
                      interfaceSignals := #statInterfaceSignalsHmi[38].valueSymbolLeft,
                      ENO => #_w1);
   IF #_w1 THEN
       #instSignals38Right(interfaceSignals := #statInterfaceSignalsHmi[38].valueSymbolRight);   // "LAF_InterfaceSignalsBool"
   END_IF;
END_REGION

REGION Network 44: Interface Signals 05 -Example: Model Flex-Pro-Line - IN/OUT- / Interface Signals 39
   // Aufruf des Schnittstellen Signal Bausteins Ba-Bereich 4 / Call the interface signals bool blocks of opmode 4
   RUNG wire#powerrail
      #instSignals39Left(signal00 := "SBK03"."ROLL CHANGE TOP SS.AUTO", signal01 := "SBK03"."ROLL CHANGE BTM SS.AUTO", signal02 := "SBK03"."ROLL CHANGE TOP SS.CHANGE", signal03 := "SBK03"."ROLL CHANGE BTM SS.CHANGE", signal04 := "SBK03"."ROLL CHANGE LH IN PROGRESS", signal05 := "SBK03"."ROLL CHANGE RH IN PROGRESS", signal06 :=, signal07 :=, signal08 :=, signal09 :=, signal10 :=, signal11 :=, signal12 :=, signal13 :=, signal14 :=, signal15 :=, interfaceSignals := #statInterfaceSignalsHmi[39].valueSymbolLeft)
      #instSignals39Right(signal00 :=, signal01 :=, signal02 :=, signal03 :=, signal04 :=, signal05 :=, signal06 :=, signal07 :=, signal08 :=, signal09 :=, signal10 :=, signal11 :=, signal12 :=, signal13 :=, signal14 :=, signal15 :=, interfaceSignals := #statInterfaceSignalsHmi[39].valueSymbolRight)
   END_RUNG
   // the same network as SCL:
   #instSignals39Left(signal00 := "SBK03"."ROLL CHANGE TOP SS.AUTO",   // "LAF_InterfaceSignalsBool"
                      signal01 := "SBK03"."ROLL CHANGE BTM SS.AUTO",
                      signal02 := "SBK03"."ROLL CHANGE TOP SS.CHANGE",
                      signal03 := "SBK03"."ROLL CHANGE BTM SS.CHANGE",
                      signal04 := "SBK03"."ROLL CHANGE LH IN PROGRESS",
                      signal05 := "SBK03"."ROLL CHANGE RH IN PROGRESS",
                      interfaceSignals := #statInterfaceSignalsHmi[39].valueSymbolLeft,
                      ENO => #_w1);
   IF #_w1 THEN
       #instSignals39Right(interfaceSignals := #statInterfaceSignalsHmi[39].valueSymbolRight);   // "LAF_InterfaceSignalsBool"
   END_IF;
END_REGION

REGION Network 45: Interface Signals 05 -Example: Model Flex-Pro-Line - IN/OUT- / Interface Signals 40
   // Aufruf des Schnittstellen Signal Bausteins Ba-Bereich 4 / Call the interface signals bool blocks of opmode 4
